KUKA KRL program: f1_Kuka_APT203T03S03.SRC

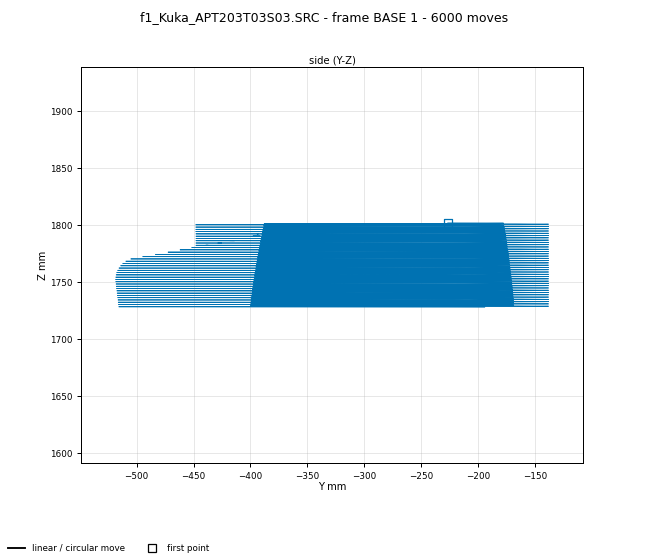
[picture p0: tool path of f1_Kuka_APT203T03S03.SRC in frame BASE 1, 6000 of 6001 moves have a stored position in this frame; points joined in program order, loops and branches not executed]
&ACCESS RVP
&REL 2
&PARAM TEMPLATE = C:\KRC\Roboter\Template\vorgabe
&PARAM EDITMASK = *
DEF f1_Kuka_APT203T03S03()


;FOLD INI;%{PE}%V3.2.0,%MKUKATPBASIS,%CINIT,%VCOMMON,%P
  ;FOLD BAS INI;%{E}%V3.2.0,%MKUKATPBASIS,%CINIT,%VINIT,%P
    GLOBAL INTERRUPT DECL 3 WHEN $STOPMESS==TRUE DO IR_STOPM ( )
    INTERRUPT ON 3
    BAS (#INITMOV,0 )
  ;ENDFOLD (BAS INI)
  ;FOLD USER INI;%{E}%V3.2.0,%MKUKATPUSER,%CINIT,%VINIT,%P
    ;Make your modifications here
  ;ENDFOLD (USER INI)
;ENDFOLD (INI)


;*** Make Null PTP Move
  PTP $pos_act

;*** Auto Load The Correct TOOL Data
  $tool=tool_data[3]

;*** Auto Load The Correct BASE Data
  $base=base_data[1]

  $ADVANCE = 5

;*** Restate Last Velocity
MMPM(30000.0)
SetRPM(6000)
LIN {X 0.049,Y -226.868,Z 1802.195,A 0.000,B 0.000,C 90.000,E1 35.105} C_DIS
LIN {X -0.089,Y -218.794,Z 1802.178,A 0.000,B 0.000,C 90.000,E1 32.084} C_DIS
LIN {X 0.015,Y -211.271,Z 1802.161,A 0.000,B 0.000,C 90.000,E1 28.949} C_DIS
LIN {X -0.003,Y -204.423,Z 1802.143,A 0.000,B 0.000,C 90.000,E1 25.796} C_DIS
LIN {X 0.008,Y -198.407,Z 1802.125,A 0.000,B 0.000,C 90.000,E1 22.589} C_DIS
LIN {X 0.076,Y -193.126,Z 1802.107,A 0.000,B 0.000,C 90.000,E1 19.322} C_DIS
LIN {X -0.059,Y -188.899,Z 1802.089,A 0.000,B 0.000,C 90.000,E1 16.079} C_DIS
LIN {X 0.063,Y -184.696,Z 1802.066,A 0.000,B 0.000,C 90.000,E1 11.895} C_DIS
LIN {X 0.091,Y -181.548,Z 1802.043,A 0.000,B 0.000,C 90.000,E1 7.701} C_DIS
LIN {X -0.028,Y -178.910,Z 1802.010,A 0.000,B 0.000,C 90.000,E1 1.835} C_DIS
LIN {X 0.066,Y -177.903,Z 1801.964,A 0.000,B 0.000,C 90.000,E1 353.571} C_DIS
LIN {X 0.025,Y -178.856,Z 1801.931,A 0.000,B 0.000,C 90.000,E1 347.645} C_DIS
LIN {X -0.075,Y -181.512,Z 1801.894,A 0.000,B 0.000,C 90.000,E1 340.913} C_DIS
LIN {X 0.004,Y -184.682,Z 1801.866,A 0.000,B 0.000,C 90.000,E1 335.845} C_DIS
LIN {X -0.006,Y -188.687,Z 1801.838,A 0.000,B 0.000,C 90.000,E1 330.845} C_DIS
LIN {X 0.009,Y -192.663,Z 1801.815,A 0.000,B 0.000,C 90.000,E1 326.707} C_DIS
LIN {X -0.078,Y -197.668,Z 1801.792,A 0.000,B 0.000,C 90.000,E1 322.637} C_DIS
LIN {X -0.028,Y -202.764,Z 1801.774,A 0.000,B 0.000,C 90.000,E1 319.380} C_DIS
LIN {X -0.078,Y -207.391,Z 1801.761,A 0.000,B 0.000,C 90.000,E1 316.986} C_DIS
LIN {X -0.051,Y -212.928,Z 1801.748,A 0.000,B 0.000,C 90.000,E1 314.595} C_DIS
LIN {X -0.018,Y -217.212,Z 1801.739,A 0.000,B 0.000,C 90.000,E1 313.014} C_DIS
LIN {X -0.070,Y -222.200,Z 1801.730,A 0.000,B 0.000,C 90.000,E1 311.472} C_DIS
LIN {X -0.065,Y -227.868,Z 1801.722,A 0.000,B 0.000,C 90.000,E1 309.930} C_DIS
LIN {X 0.041,Y -234.269,Z 1801.713,A 0.000,B 0.000,C 90.000,E1 308.382} C_DIS
LIN {X 0.068,Y -243.180,Z 1801.703,A 0.000,B 0.000,C 90.000,E1 306.503} C_DIS
LIN {X -0.042,Y -255.247,Z 1801.691,A 0.000,B 0.000,C 90.000,E1 304.326} C_DIS
LIN {X 0.152,Y -268.384,Z 1801.679,A 0.000,B 0.000,C 90.000,E1 302.133} C_DIS
LIN {X -0.140,Y -287.357,Z 1801.663,A 0.000,B 0.000,C 90.000,E1 299.411} C_DIS
LIN {X 0.029,Y -307.519,Z 1801.648,A 0.000,B 0.000,C 90.000,E1 296.693} C_DIS
LIN {X -0.125,Y -323.073,Z 1801.637,A 0.000,B 0.000,C 90.000,E1 294.771} C_DIS
LIN {X 0.059,Y -335.908,Z 1801.629,A 0.000,B 0.000,C 90.000,E1 293.153} C_DIS
LIN {X 0.152,Y -348.343,Z 1801.620,A 0.000,B 0.000,C 90.000,E1 291.589} C_DIS
LIN {X 0.091,Y -355.528,Z 1801.615,A 0.000,B 0.000,C 90.000,E1 290.684} C_DIS
LIN {X -0.107,Y -362.258,Z 1801.610,A 0.000,B 0.000,C 90.000,E1 289.812} C_DIS
LIN {X -0.036,Y -368.425,Z 1801.605,A 0.000,B 0.000,C 90.000,E1 288.906} C_DIS
LIN {X 0.103,Y -373.893,Z 1801.600,A 0.000,B 0.000,C 90.000,E1 288.000} C_DIS
LIN {X -0.069,Y -378.389,Z 1801.595,A 0.000,B 0.000,C 90.000,E1 287.149} C_DIS
LIN {X 0.054,Y -381.951,Z 1801.590,A 0.000,B 0.000,C 90.000,E1 286.260} C_DIS
LIN {X -0.158,Y -384.694,Z 1801.586,A 0.000,B 0.000,C 90.000,E1 285.426} C_DIS
LIN {X -0.008,Y -386.071,Z 1801.582,A 0.000,B 0.000,C 90.000,E1 284.828} C_DIS
LIN {X 0.056,Y -387.102,Z 1801.579,A 0.000,B 0.000,C 90.000,E1 284.245} C_DIS
LIN {X -0.153,Y -387.749,Z 1801.576,A 0.000,B 0.000,C 90.000,E1 283.703} C_DIS
LIN {X -0.072,Y -388.016,Z 1801.573,A 0.000,B 0.000,C 90.000,E1 283.119} C_DIS
LIN {X 0.015,Y -387.896,Z 1801.570,A 0.000,B 0.000,C 90.000,E1 282.535} C_DIS
LIN {X 0.105,Y -387.385,Z 1801.567,A 0.000,B 0.000,C 90.000,E1 281.951} C_DIS
LIN {X -0.184,Y -386.489,Z 1801.563,A 0.000,B 0.000,C 90.000,E1 281.422} C_DIS
LIN {X -0.097,Y -385.220,Z 1801.560,A 0.000,B 0.000,C 90.000,E1 280.838} C_DIS
LIN {X -0.016,Y -383.567,Z 1801.557,A 0.000,B 0.000,C 90.000,E1 280.254} C_DIS
LIN {X 0.084,Y -380.530,Z 1801.552,A 0.000,B 0.000,C 90.000,E1 279.378} C_DIS
LIN {X 0.091,Y -376.860,Z 1801.547,A 0.000,B 0.000,C 90.000,E1 278.511} C_DIS
LIN {X 0.061,Y -374.045,Z 1801.544,A 0.000,B 0.000,C 90.000,E1 277.936} C_DIS
LIN {X 0.013,Y -369.161,Z 1801.539,A 0.000,B 0.000,C 90.000,E1 277.068} C_DIS
LIN {X -0.074,Y -363.286,Z 1801.534,A 0.000,B 0.000,C 90.000,E1 276.201} C_DIS
LIN {X -0.174,Y -358.718,Z 1801.531,A 0.000,B 0.000,C 90.000,E1 275.625} C_DIS
LIN {X 0.056,Y -353.637,Z 1801.528,A 0.000,B 0.000,C 90.000,E1 274.992} C_DIS
LIN {X -0.079,Y -347.942,Z 1801.524,A 0.000,B 0.000,C 90.000,E1 274.416} C_DIS
LIN {X 0.034,Y -342.104,Z 1801.521,A 0.000,B 0.000,C 90.000,E1 273.841} C_DIS
LIN {X 0.014,Y -336.087,Z 1801.518,A 0.000,B 0.000,C 90.000,E1 273.326} C_DIS
LIN {X -0.054,Y -330.045,Z 1801.516,A 0.000,B 0.000,C 90.000,E1 272.865} C_DIS
LIN {X 0.000,Y -323.550,Z 1801.513,A 0.000,B 0.000,C 90.000,E1 272.407} C_DIS
LIN {X -0.005,Y -316.745,Z 1801.511,A 0.000,B 0.000,C 90.000,E1 272.007} C_DIS
LIN {X -0.014,Y -309.834,Z 1801.509,A 0.000,B 0.000,C 90.000,E1 271.661} C_DIS
LIN {X -0.059,Y -302.584,Z 1801.508,A 0.000,B 0.000,C 90.000,E1 271.375} C_DIS
LIN {X -0.122,Y -294.791,Z 1801.506,A 0.000,B 0.000,C 90.000,E1 271.146} C_DIS
LIN {X -0.005,Y -284.000,Z 1801.505,A 0.000,B 0.000,C 90.000,E1 270.859} C_DIS
LIN {X 0.024,Y -272.702,Z 1801.504,A 0.000,B 0.000,C 90.000,E1 270.630} C_DIS
LIN {X -0.103,Y -257.783,Z 1801.502,A 0.000,B 0.000,C 90.000,E1 270.401} C_DIS
LIN {X 0.105,Y -246.724,Z 1801.501,A 0.000,B 0.000,C 90.000,E1 270.229} C_DIS
LIN {X 0.009,Y -235.036,Z 1801.501,A 0.000,B 0.000,C 90.000,E1 270.172} C_DIS
LIN {X -0.015,Y -181.579,Z 1801.501,A 0.000,B 0.000,C 90.000,E1 270.172} C_DIS
LIN {X -0.048,Y -180.792,Z 1801.471,A 0.000,B 0.000,C 90.000,E1 264.780} C_DIS
LIN {X 0.026,Y -178.891,Z 1801.443,A 0.000,B 0.000,C 90.000,E1 259.690} C_DIS
LIN {X -0.068,Y -175.934,Z 1801.414,A 0.000,B 0.000,C 90.000,E1 254.629} C_DIS
LIN {X 0.048,Y -175.381,Z 1801.410,A 0.000,B 0.000,C 90.000,E1 253.740} C_DIS
LIN {X 0.045,Y -172.154,Z 1801.386,A 0.000,B 0.000,C 90.000,E1 249.464} C_DIS
LIN {X 0.082,Y -171.621,Z 1801.381,A 0.000,B 0.000,C 90.000,E1 248.592} C_DIS
LIN {X 0.069,Y -167.843,Z 1801.357,A 0.000,B 0.000,C 90.000,E1 244.280} C_DIS
LIN {X 0.010,Y -166.572,Z 1801.348,A 0.000,B 0.000,C 90.000,E1 242.564} C_DIS
LIN {X -0.004,Y -162.565,Z 1801.323,A 0.000,B 0.000,C 90.000,E1 238.201} C_DIS
LIN {X 0.056,Y -161.246,Z 1801.314,A 0.000,B 0.000,C 90.000,E1 236.421} C_DIS
LIN {X -0.034,Y -157.249,Z 1801.289,A 0.000,B 0.000,C 90.000,E1 232.029} C_DIS
LIN {X 0.013,Y -155.972,Z 1801.279,A 0.000,B 0.000,C 90.000,E1 230.231} C_DIS
LIN {X 0.071,Y -152.226,Z 1801.254,A 0.000,B 0.000,C 90.000,E1 225.729} C_DIS
LIN {X -0.019,Y -150.469,Z 1801.239,A 0.000,B 0.000,C 90.000,E1 223.056} C_DIS
LIN {X 0.001,Y -147.194,Z 1801.214,A 0.000,B 0.000,C 90.000,E1 218.508} C_DIS
LIN {X 0.082,Y -145.213,Z 1801.194,A 0.000,B 0.000,C 90.000,E1 214.818} C_DIS
LIN {X -0.008,Y -142.345,Z 1801.163,A 0.000,B 0.000,C 90.000,E1 209.333} C_DIS
LIN {X 0.045,Y -141.733,Z 1801.153,A 0.000,B 0.000,C 90.000,E1 207.462} C_DIS
LIN {X 0.027,Y -139.483,Z 1801.117,A 0.000,B 0.000,C 90.000,E1 200.972} C_DIS
LIN {X 0.015,Y -138.984,Z 1801.101,A 0.000,B 0.000,C 90.000,E1 198.181} C_DIS
LIN {X -0.023,Y -138.333,Z 1801.054,A 0.000,B 0.000,C 90.000,E1 189.792} C_DIS
LIN {X 0.001,Y -139.425,Z 1801.008,A 0.000,B 0.000,C 90.000,E1 181.375} C_DIS
LIN {X 0.055,Y -141.349,Z 1800.971,A 0.000,B 0.000,C 90.000,E1 174.837} C_DIS
LIN {X 0.032,Y -142.703,Z 1800.956,A 0.000,B 0.000,C 90.000,E1 172.064} C_DIS
LIN {X -0.009,Y -145.073,Z 1800.930,A 0.000,B 0.000,C 90.000,E1 167.465} C_DIS
LIN {X -0.013,Y -147.698,Z 1800.910,A 0.000,B 0.000,C 90.000,E1 163.795} C_DIS
LIN {X 0.019,Y -150.349,Z 1800.890,A 0.000,B 0.000,C 90.000,E1 160.134} C_DIS
LIN {X 0.013,Y -154.604,Z 1800.865,A 0.000,B 0.000,C 90.000,E1 155.613} C_DIS
LIN {X 0.019,Y -158.145,Z 1800.845,A 0.000,B 0.000,C 90.000,E1 152.025} C_DIS
LIN {X 0.065,Y -162.432,Z 1800.825,A 0.000,B 0.000,C 90.000,E1 148.456} C_DIS
LIN {X -0.039,Y -166.691,Z 1800.805,A 0.000,B 0.000,C 90.000,E1 144.975} C_DIS
LIN {X 0.074,Y -171.697,Z 1800.786,A 0.000,B 0.000,C 90.000,E1 141.457} C_DIS
LIN {X 0.008,Y -176.669,Z 1800.767,A 0.000,B 0.000,C 90.000,E1 138.038} C_DIS
LIN {X 0.003,Y -180.965,Z 1800.753,A 0.000,B 0.000,C 90.000,E1 135.486} C_DIS
LIN {X -0.010,Y -186.388,Z 1800.734,A 0.000,B 0.000,C 90.000,E1 132.123} C_DIS
LIN {X -0.070,Y -191.018,Z 1800.720,A 0.000,B 0.000,C 90.000,E1 129.644} C_DIS
LIN {X 0.123,Y -196.798,Z 1800.702,A 0.000,B 0.000,C 90.000,E1 126.297} C_DIS
LIN {X 0.042,Y -200.050,Z 1800.693,A 0.000,B 0.000,C 90.000,E1 124.692} C_DIS
LIN {X 0.036,Y -207.551,Z 1800.670,A 0.000,B 0.000,C 90.000,E1 120.669} C_DIS
LIN {X 0.040,Y -210.761,Z 1800.662,A 0.000,B 0.000,C 90.000,E1 119.077} C_DIS
LIN {X 0.079,Y -213.754,Z 1800.652,A 0.000,B 0.000,C 90.000,E1 117.385} C_DIS
LIN {X 0.074,Y -337.789,Z 1800.652,A 0.000,B 0.000,C 90.000,E1 117.385} C_DIS
LIN {X 0.022,Y -338.618,Z 1800.652,A 0.000,B 0.000,C 90.000,E1 117.385} C_DIS
LIN {X 0.019,Y -343.715,Z 1800.650,A 0.000,B 0.000,C 90.000,E1 117.052} C_DIS
LIN {X -0.141,Y -345.694,Z 1800.648,A 0.000,B 0.000,C 90.000,E1 116.744} C_DIS
LIN {X 0.023,Y -347.535,Z 1800.645,A 0.000,B 0.000,C 90.000,E1 116.104} C_DIS
LIN {X 0.201,Y -349.007,Z 1800.642,A 0.000,B 0.000,C 90.000,E1 115.463} C_DIS
LIN {X -0.076,Y -350.263,Z 1800.638,A 0.000,B 0.000,C 90.000,E1 114.899} C_DIS
LIN {X 0.121,Y -351.140,Z 1800.635,A 0.000,B 0.000,C 90.000,E1 114.259} C_DIS
LIN {X -0.140,Y -351.151,Z 1800.631,A 0.000,B 0.000,C 90.000,E1 113.695} C_DIS
LIN {X 0.111,Y -343.512,Z 1800.608,A 0.000,B 0.000,C 90.000,E1 109.396} C_DIS
LIN {X -0.001,Y -337.369,Z 1800.580,A 0.000,B 0.000,C 90.000,E1 104.411} C_DIS
LIN {X -0.058,Y -337.416,Z 1800.580,A 0.000,B 0.000,C 90.000,E1 104.411} C_DIS
LIN {X -0.125,Y -354.092,Z 1800.568,A 0.000,B 0.000,C 90.000,E1 102.355} C_DIS
LIN {X -0.015,Y -372.554,Z 1800.557,A 0.000,B 0.000,C 90.000,E1 100.310} C_DIS
LIN {X 0.103,Y -391.414,Z 1800.547,A 0.000,B 0.000,C 90.000,E1 98.454} C_DIS
LIN {X 0.110,Y -410.686,Z 1800.538,A 0.000,B 0.000,C 90.000,E1 96.777} C_DIS
LIN {X 0.041,Y -433.088,Z 1800.528,A 0.000,B 0.000,C 90.000,E1 95.049} C_DIS
LIN {X 0.018,Y -438.722,Z 1800.526,A 0.000,B 0.000,C 90.000,E1 94.645} C_DIS
LIN {X -0.017,Y -442.704,Z 1800.524,A 0.000,B 0.000,C 90.000,E1 94.245} C_DIS
LIN {X -0.198,Y -444.401,Z 1800.522,A 0.000,B 0.000,C 90.000,E1 94.012} C_DIS
LIN {X 0.033,Y -445.693,Z 1800.521,A 0.000,B 0.000,C 90.000,E1 93.726} C_DIS
LIN {X -0.045,Y -447.394,Z 1800.518,A 0.000,B 0.000,C 90.000,E1 93.212} C_DIS
LIN {X -0.092,Y -448.057,Z 1800.515,A 0.000,B 0.000,C 90.000,E1 92.694} C_DIS
LIN {X -0.150,Y -447.790,Z 1800.512,A 0.000,B 0.000,C 90.000,E1 92.178} C_DIS
LIN {X -0.188,Y -446.557,Z 1800.509,A 0.000,B 0.000,C 90.000,E1 91.661} C_DIS
LIN {X 0.009,Y -445.523,Z 1800.508,A 0.000,B 0.000,C 90.000,E1 91.375} C_DIS
LIN {X 0.203,Y -444.146,Z 1800.506,A 0.000,B 0.000,C 90.000,E1 91.088} C_DIS
LIN {X -0.166,Y -430.943,Z 1800.495,A 0.000,B 0.000,C 90.000,E1 89.026} C_DIS
LIN {X -0.194,Y -420.924,Z 1800.485,A 0.000,B 0.000,C 90.000,E1 87.421} C_DIS
LIN {X 0.117,Y -409.108,Z 1800.475,A 0.000,B 0.000,C 90.000,E1 85.469} C_DIS
LIN {X -0.190,Y -397.220,Z 1800.464,A 0.000,B 0.000,C 90.000,E1 83.571} C_DIS
LIN {X 0.131,Y -385.260,Z 1800.453,A 0.000,B 0.000,C 90.000,E1 81.546} C_DIS
LIN {X -0.109,Y -373.304,Z 1800.442,A 0.000,B 0.000,C 90.000,E1 79.567} C_DIS
LIN {X 0.097,Y -356.843,Z 1800.426,A 0.000,B 0.000,C 90.000,E1 76.589} C_DIS
LIN {X -0.096,Y -355.062,Z 1800.424,A 0.000,B 0.000,C 90.000,E1 76.284} C_DIS
LIN {X 0.190,Y -355.058,Z 1800.424,A 0.000,B 0.000,C 90.000,E1 76.228} C_DIS
LIN {X -0.055,Y -360.061,Z 1800.412,A 0.000,B 0.000,C 90.000,E1 74.212} C_DIS
LIN {X -0.056,Y -360.127,Z 1800.409,A 0.000,B 0.000,C 90.000,E1 73.614} C_DIS
LIN {X -0.047,Y -359.374,Z 1800.406,A 0.000,B 0.000,C 90.000,E1 73.015} C_DIS
LIN {X -0.038,Y -358.243,Z 1800.402,A 0.000,B 0.000,C 90.000,E1 72.417} C_DIS
LIN {X -0.041,Y -355.353,Z 1800.396,A 0.000,B 0.000,C 90.000,E1 71.221} C_DIS
LIN {X 0.033,Y -351.986,Z 1800.389,A 0.000,B 0.000,C 90.000,E1 70.007} C_DIS
LIN {X -0.070,Y -346.491,Z 1800.379,A 0.000,B 0.000,C 90.000,E1 68.209} C_DIS
LIN {X 0.051,Y -340.599,Z 1800.369,A 0.000,B 0.000,C 90.000,E1 66.357} C_DIS
LIN {X -0.119,Y -334.493,Z 1800.358,A 0.000,B 0.000,C 90.000,E1 64.537} C_DIS
LIN {X -0.105,Y -328.066,Z 1800.348,A 0.000,B 0.000,C 90.000,E1 62.666} C_DIS
LIN {X 0.119,Y -322.241,Z 1800.339,A 0.000,B 0.000,C 90.000,E1 61.051} C_DIS
LIN {X 0.118,Y -315.910,Z 1800.330,A 0.000,B 0.000,C 90.000,E1 59.459} C_DIS
LIN {X 0.068,Y -307.744,Z 1800.320,A 0.000,B 0.000,C 90.000,E1 57.533} C_DIS
LIN {X -0.060,Y -299.204,Z 1800.309,A 0.000,B 0.000,C 90.000,E1 55.595} C_DIS
LIN {X 0.066,Y -290.532,Z 1800.298,A 0.000,B 0.000,C 90.000,E1 53.577} C_DIS
LIN {X -0.007,Y -279.032,Z 1800.283,A 0.000,B 0.000,C 90.000,E1 50.884} C_DIS
LIN {X 0.046,Y -266.931,Z 1800.265,A 0.000,B 0.000,C 90.000,E1 47.757} C_DIS
LIN {X -0.061,Y -255.644,Z 1800.248,A 0.000,B 0.000,C 90.000,E1 44.595} C_DIS
LIN {X 0.060,Y -246.134,Z 1800.232,A 0.000,B 0.000,C 90.000,E1 41.676} C_DIS
LIN {X -0.019,Y -236.966,Z 1800.215,A 0.000,B 0.000,C 90.000,E1 38.749} C_DIS
LIN {X 0.044,Y -226.156,Z 1800.194,A 0.000,B 0.000,C 90.000,E1 34.978} C_DIS
LIN {X 0.009,Y -218.086,Z 1800.177,A 0.000,B 0.000,C 90.000,E1 31.926} C_DIS
LIN {X -0.017,Y -210.578,Z 1800.160,A 0.000,B 0.000,C 90.000,E1 28.821} C_DIS
LIN {X -0.051,Y -203.742,Z 1800.143,A 0.000,B 0.000,C 90.000,E1 25.668} C_DIS
LIN {X -0.056,Y -197.761,Z 1800.125,A 0.000,B 0.000,C 90.000,E1 22.461} C_DIS
LIN {X -0.069,Y -192.520,Z 1800.107,A 0.000,B 0.000,C 90.000,E1 19.214} C_DIS
LIN {X 0.025,Y -188.325,Z 1800.088,A 0.000,B 0.000,C 90.000,E1 15.898} C_DIS
LIN {X -0.055,Y -184.173,Z 1800.065,A 0.000,B 0.000,C 90.000,E1 11.771} C_DIS
LIN {X -0.074,Y -181.053,Z 1800.042,A 0.000,B 0.000,C 90.000,E1 7.587} C_DIS
LIN {X 0.014,Y -178.233,Z 1800.005,A 0.000,B 0.000,C 90.000,E1 0.802} C_DIS
LIN {X 0.050,Y -177.541,Z 1799.964,A 0.000,B 0.000,C 90.000,E1 353.571} C_DIS
LIN {X -0.093,Y -178.758,Z 1799.927,A 0.000,B 0.000,C 90.000,E1 346.825} C_DIS
LIN {X 0.047,Y -181.197,Z 1799.894,A 0.000,B 0.000,C 90.000,E1 340.859} C_DIS
LIN {X -0.056,Y -184.377,Z 1799.866,A 0.000,B 0.000,C 90.000,E1 335.845} C_DIS
LIN {X 0.086,Y -188.424,Z 1799.838,A 0.000,B 0.000,C 90.000,E1 330.795} C_DIS
LIN {X -0.073,Y -192.446,Z 1799.815,A 0.000,B 0.000,C 90.000,E1 326.707} C_DIS
LIN {X 0.108,Y -197.548,Z 1799.792,A 0.000,B 0.000,C 90.000,E1 322.557} C_DIS
LIN {X 0.009,Y -201.339,Z 1799.779,A 0.000,B 0.000,C 90.000,E1 320.150} C_DIS
LIN {X 0.082,Y -205.789,Z 1799.765,A 0.000,B 0.000,C 90.000,E1 317.715} C_DIS
LIN {X 0.079,Y -211.070,Z 1799.752,A 0.000,B 0.000,C 90.000,E1 315.324} C_DIS
LIN {X -0.019,Y -216.221,Z 1799.741,A 0.000,B 0.000,C 90.000,E1 313.380} C_DIS
LIN {X -0.089,Y -221.080,Z 1799.732,A 0.000,B 0.000,C 90.000,E1 311.838} C_DIS
LIN {X 0.075,Y -226.607,Z 1799.724,A 0.000,B 0.000,C 90.000,E1 310.253} C_DIS
LIN {X -0.010,Y -232.839,Z 1799.715,A 0.000,B 0.000,C 90.000,E1 308.749} C_DIS
LIN {X -0.013,Y -241.593,Z 1799.705,A 0.000,B 0.000,C 90.000,E1 306.870} C_DIS
LIN {X -0.012,Y -253.471,Z 1799.693,A 0.000,B 0.000,C 90.000,E1 304.659} C_DIS
LIN {X 0.053,Y -268.761,Z 1799.679,A 0.000,B 0.000,C 90.000,E1 302.133} C_DIS
LIN {X 0.156,Y -287.772,Z 1799.663,A 0.000,B 0.000,C 90.000,E1 299.333} C_DIS
LIN {X -0.030,Y -307.933,Z 1799.648,A 0.000,B 0.000,C 90.000,E1 296.693} C_DIS
LIN {X -0.145,Y -323.490,Z 1799.637,A 0.000,B 0.000,C 90.000,E1 294.771} C_DIS
LIN {X 0.061,Y -336.326,Z 1799.629,A 0.000,B 0.000,C 90.000,E1 293.153} C_DIS
LIN {X 0.162,Y -348.781,Z 1799.620,A 0.000,B 0.000,C 90.000,E1 291.589} C_DIS
LIN {X -0.186,Y -358.269,Z 1799.613,A 0.000,B 0.000,C 90.000,E1 290.429} C_DIS
LIN {X -0.033,Y -364.845,Z 1799.608,A 0.000,B 0.000,C 90.000,E1 289.504} C_DIS
LIN {X 0.070,Y -370.827,Z 1799.603,A 0.000,B 0.000,C 90.000,E1 288.598} C_DIS
LIN {X 0.131,Y -374.380,Z 1799.600,A 0.000,B 0.000,C 90.000,E1 288.000} C_DIS
LIN {X -0.141,Y -377.473,Z 1799.597,A 0.000,B 0.000,C 90.000,E1 287.457} C_DIS
LIN {X 0.078,Y -381.323,Z 1799.592,A 0.000,B 0.000,C 90.000,E1 286.551} C_DIS
LIN {X 0.106,Y -383.392,Z 1799.589,A 0.000,B 0.000,C 90.000,E1 285.969} C_DIS
LIN {X -0.116,Y -385.134,Z 1799.586,A 0.000,B 0.000,C 90.000,E1 285.426} C_DIS
LIN {X 0.038,Y -386.506,Z 1799.582,A 0.000,B 0.000,C 90.000,E1 284.828} C_DIS
LIN {X 0.104,Y -387.522,Z 1799.579,A 0.000,B 0.000,C 90.000,E1 284.245} C_DIS
LIN {X -0.103,Y -388.189,Z 1799.576,A 0.000,B 0.000,C 90.000,E1 283.703} C_DIS
LIN {X -0.020,Y -388.450,Z 1799.573,A 0.000,B 0.000,C 90.000,E1 283.119} C_DIS
LIN {X 0.070,Y -388.333,Z 1799.570,A 0.000,B 0.000,C 90.000,E1 282.535} C_DIS
LIN {X 0.163,Y -387.840,Z 1799.567,A 0.000,B 0.000,C 90.000,E1 281.951} C_DIS
LIN {X -0.124,Y -386.939,Z 1799.563,A 0.000,B 0.000,C 90.000,E1 281.422} C_DIS
LIN {X -0.035,Y -385.696,Z 1799.560,A 0.000,B 0.000,C 90.000,E1 280.838} C_DIS
LIN {X 0.049,Y -384.051,Z 1799.557,A 0.000,B 0.000,C 90.000,E1 280.254} C_DIS
LIN {X 0.153,Y -381.043,Z 1799.552,A 0.000,B 0.000,C 90.000,E1 279.378} C_DIS
LIN {X 0.165,Y -377.390,Z 1799.547,A 0.000,B 0.000,C 90.000,E1 278.511} C_DIS
LIN {X 0.137,Y -374.564,Z 1799.544,A 0.000,B 0.000,C 90.000,E1 277.936} C_DIS
LIN {X 0.092,Y -369.645,Z 1799.539,A 0.000,B 0.000,C 90.000,E1 277.068} C_DIS
LIN {X 0.008,Y -363.751,Z 1799.534,A 0.000,B 0.000,C 90.000,E1 276.201} C_DIS
LIN {X -0.134,Y -356.711,Z 1799.530,A 0.000,B 0.000,C 90.000,E1 275.334} C_DIS
LIN {X 0.110,Y -351.326,Z 1799.526,A 0.000,B 0.000,C 90.000,E1 274.702} C_DIS
LIN {X 0.100,Y -345.622,Z 1799.523,A 0.000,B 0.000,C 90.000,E1 274.131} C_DIS
LIN {X 0.001,Y -339.711,Z 1799.520,A 0.000,B 0.000,C 90.000,E1 273.612} C_DIS
LIN {X 0.107,Y -333.582,Z 1799.517,A 0.000,B 0.000,C 90.000,E1 273.094} C_DIS
LIN {X 0.074,Y -327.302,Z 1799.515,A 0.000,B 0.000,C 90.000,E1 272.636} C_DIS
LIN {X -0.055,Y -320.739,Z 1799.512,A 0.000,B 0.000,C 90.000,E1 272.236} C_DIS
LIN {X 0.073,Y -313.919,Z 1799.510,A 0.000,B 0.000,C 90.000,E1 271.835} C_DIS
LIN {X -0.130,Y -306.791,Z 1799.508,A 0.000,B 0.000,C 90.000,E1 271.547} C_DIS
LIN {X -0.041,Y -299.284,Z 1799.507,A 0.000,B 0.000,C 90.000,E1 271.260} C_DIS
LIN {X -0.136,Y -287.817,Z 1799.505,A 0.000,B 0.000,C 90.000,E1 270.974} C_DIS
LIN {X 0.131,Y -277.007,Z 1799.504,A 0.000,B 0.000,C 90.000,E1 270.688} C_DIS
LIN {X -0.076,Y -257.992,Z 1799.502,A 0.000,B 0.000,C 90.000,E1 270.401} C_DIS
LIN {X 0.118,Y -246.142,Z 1799.501,A 0.000,B 0.000,C 90.000,E1 270.229} C_DIS
LIN {X 0.034,Y -233.356,Z 1799.501,A 0.000,B 0.000,C 90.000,E1 270.172} C_DIS
LIN {X 0.006,Y -181.579,Z 1799.501,A 0.000,B 0.000,C 90.000,E1 270.172} C_DIS
LIN {X -0.023,Y -180.795,Z 1799.471,A 0.000,B 0.000,C 90.000,E1 264.780} C_DIS
LIN {X 0.051,Y -178.894,Z 1799.443,A 0.000,B 0.000,C 90.000,E1 259.690} C_DIS
LIN {X -0.044,Y -175.937,Z 1799.415,A 0.000,B 0.000,C 90.000,E1 254.629} C_DIS
LIN {X 0.070,Y -175.388,Z 1799.410,A 0.000,B 0.000,C 90.000,E1 253.740} C_DIS
LIN {X -0.093,Y -172.159,Z 1799.386,A 0.000,B 0.000,C 90.000,E1 249.518} C_DIS
LIN {X -0.054,Y -171.627,Z 1799.381,A 0.000,B 0.000,C 90.000,E1 248.646} C_DIS
LIN {X -0.058,Y -167.850,Z 1799.357,A 0.000,B 0.000,C 90.000,E1 244.332} C_DIS
LIN {X 0.033,Y -166.579,Z 1799.348,A 0.000,B 0.000,C 90.000,E1 242.564} C_DIS
LIN {X 0.019,Y -162.571,Z 1799.323,A 0.000,B 0.000,C 90.000,E1 238.201} C_DIS
LIN {X 0.078,Y -161.253,Z 1799.314,A 0.000,B 0.000,C 90.000,E1 236.421} C_DIS
LIN {X -0.012,Y -157.255,Z 1799.289,A 0.000,B 0.000,C 90.000,E1 232.029} C_DIS
LIN {X 0.035,Y -155.977,Z 1799.279,A 0.000,B 0.000,C 90.000,E1 230.231} C_DIS
LIN {X 0.092,Y -152.232,Z 1799.254,A 0.000,B 0.000,C 90.000,E1 225.729} C_DIS
LIN {X 0.003,Y -150.474,Z 1799.239,A 0.000,B 0.000,C 90.000,E1 223.056} C_DIS
LIN {X -0.069,Y -147.199,Z 1799.214,A 0.000,B 0.000,C 90.000,E1 218.543} C_DIS
LIN {X -0.015,Y -145.219,Z 1799.194,A 0.000,B 0.000,C 90.000,E1 214.865} C_DIS
LIN {X 0.013,Y -142.348,Z 1799.163,A 0.000,B 0.000,C 90.000,E1 209.333} C_DIS
LIN {X -0.060,Y -141.736,Z 1799.153,A 0.000,B 0.000,C 90.000,E1 207.513} C_DIS
LIN {X 0.048,Y -139.485,Z 1799.117,A 0.000,B 0.000,C 90.000,E1 200.972} C_DIS
LIN {X 0.037,Y -138.986,Z 1799.101,A 0.000,B 0.000,C 90.000,E1 198.181} C_DIS
LIN {X -0.002,Y -138.334,Z 1799.054,A 0.000,B 0.000,C 90.000,E1 189.792} C_DIS
LIN {X 0.022,Y -139.423,Z 1799.008,A 0.000,B 0.000,C 90.000,E1 181.375} C_DIS
LIN {X -0.065,Y -141.345,Z 1798.971,A 0.000,B 0.000,C 90.000,E1 174.894} C_DIS
LIN {X 0.052,Y -142.699,Z 1798.956,A 0.000,B 0.000,C 90.000,E1 172.064} C_DIS
LIN {X 0.012,Y -145.068,Z 1798.930,A 0.000,B 0.000,C 90.000,E1 167.465} C_DIS
LIN {X 0.008,Y -147.693,Z 1798.910,A 0.000,B 0.000,C 90.000,E1 163.795} C_DIS
LIN {X 0.041,Y -150.343,Z 1798.890,A 0.000,B 0.000,C 90.000,E1 160.134} C_DIS
LIN {X 0.035,Y -154.597,Z 1798.865,A 0.000,B 0.000,C 90.000,E1 155.613} C_DIS
LIN {X 0.043,Y -158.136,Z 1798.845,A 0.000,B 0.000,C 90.000,E1 152.025} C_DIS
LIN {X 0.002,Y -162.423,Z 1798.825,A 0.000,B 0.000,C 90.000,E1 148.486} C_DIS
LIN {X -0.016,Y -166.680,Z 1798.805,A 0.000,B 0.000,C 90.000,E1 144.975} C_DIS
LIN {X 0.097,Y -171.686,Z 1798.786,A 0.000,B 0.000,C 90.000,E1 141.457} C_DIS
LIN {X -0.099,Y -176.656,Z 1798.767,A 0.000,B 0.000,C 90.000,E1 138.081} C_DIS
LIN {X 0.028,Y -180.953,Z 1798.753,A 0.000,B 0.000,C 90.000,E1 135.486} C_DIS
LIN {X 0.016,Y -186.375,Z 1798.734,A 0.000,B 0.000,C 90.000,E1 132.123} C_DIS
LIN {X -0.044,Y -191.006,Z 1798.720,A 0.000,B 0.000,C 90.000,E1 129.644} C_DIS
LIN {X -0.009,Y -196.783,Z 1798.702,A 0.000,B 0.000,C 90.000,E1 126.343} C_DIS
LIN {X 0.067,Y -200.035,Z 1798.693,A 0.000,B 0.000,C 90.000,E1 124.692} C_DIS
LIN {X 0.062,Y -207.536,Z 1798.671,A 0.000,B 0.000,C 90.000,E1 120.669} C_DIS
LIN {X 0.066,Y -210.748,Z 1798.662,A 0.000,B 0.000,C 90.000,E1 119.077} C_DIS
LIN {X 0.012,Y -212.937,Z 1798.655,A 0.000,B 0.000,C 90.000,E1 117.847} C_DIS
LIN {X -0.034,Y -337.533,Z 1798.655,A 0.000,B 0.000,C 90.000,E1 117.847} C_DIS
LIN {X 0.219,Y -342.455,Z 1798.654,A 0.000,B 0.000,C 90.000,E1 117.641} C_DIS
LIN {X 0.009,Y -344.383,Z 1798.653,A 0.000,B 0.000,C 90.000,E1 117.513} C_DIS
LIN {X 0.190,Y -347.661,Z 1798.650,A 0.000,B 0.000,C 90.000,E1 117.001} C_DIS
LIN {X -0.115,Y -348.868,Z 1798.648,A 0.000,B 0.000,C 90.000,E1 116.744} C_DIS
LIN {X -0.019,Y -353.641,Z 1798.640,A 0.000,B 0.000,C 90.000,E1 115.207} C_DIS
LIN {X -0.048,Y -357.092,Z 1798.633,A 0.000,B 0.000,C 90.000,E1 114.003} C_DIS
LIN {X 0.046,Y -358.556,Z 1798.630,A 0.000,B 0.000,C 90.000,E1 113.387} C_DIS
LIN {X 0.153,Y -359.679,Z 1798.627,A 0.000,B 0.000,C 90.000,E1 112.770} C_DIS
LIN {X -0.063,Y -360.092,Z 1798.623,A 0.000,B 0.000,C 90.000,E1 112.206} C_DIS
LIN {X 0.185,Y -358.033,Z 1798.617,A 0.000,B 0.000,C 90.000,E1 110.972} C_DIS
LIN {X -0.090,Y -350.927,Z 1798.590,A 0.000,B 0.000,C 90.000,E1 106.205} C_DIS
LIN {X 0.164,Y -347.841,Z 1798.573,A 0.000,B 0.000,C 90.000,E1 103.063} C_DIS
LIN {X 0.107,Y -347.835,Z 1798.573,A 0.000,B 0.000,C 90.000,E1 103.063} C_DIS
LIN {X -0.026,Y -365.342,Z 1798.562,A 0.000,B 0.000,C 90.000,E1 101.074} C_DIS
LIN {X 0.050,Y -384.081,Z 1798.551,A 0.000,B 0.000,C 90.000,E1 99.151} C_DIS
LIN {X 0.101,Y -403.178,Z 1798.541,A 0.000,B 0.000,C 90.000,E1 97.409} C_DIS
LIN {X -0.006,Y -425.444,Z 1798.531,A 0.000,B 0.000,C 90.000,E1 95.625} C_DIS
LIN {X 0.005,Y -439.444,Z 1798.526,A 0.000,B 0.000,C 90.000,E1 94.588} C_DIS
LIN {X -0.110,Y -443.201,Z 1798.523,A 0.000,B 0.000,C 90.000,E1 94.188} C_DIS
LIN {X 0.088,Y -444.820,Z 1798.522,A 0.000,B 0.000,C 90.000,E1 93.898} C_DIS
LIN {X -0.190,Y -446.041,Z 1798.520,A 0.000,B 0.000,C 90.000,E1 93.669} C_DIS
LIN {X 0.205,Y -447.555,Z 1798.517,A 0.000,B 0.000,C 90.000,E1 93.094} C_DIS
LIN {X 0.137,Y -448.062,Z 1798.514,A 0.000,B 0.000,C 90.000,E1 92.579} C_DIS
LIN {X 0.080,Y -447.642,Z 1798.511,A 0.000,B 0.000,C 90.000,E1 92.064} C_DIS
LIN {X 0.041,Y -446.237,Z 1798.509,A 0.000,B 0.000,C 90.000,E1 91.547} C_DIS
LIN {X -0.209,Y -445.097,Z 1798.507,A 0.000,B 0.000,C 90.000,E1 91.318} C_DIS
LIN {X -0.081,Y -440.281,Z 1798.503,A 0.000,B 0.000,C 90.000,E1 90.516} C_DIS
LIN {X 0.186,Y -428.729,Z 1798.493,A 0.000,B 0.000,C 90.000,E1 88.625} C_DIS
LIN {X -0.177,Y -416.978,Z 1798.482,A 0.000,B 0.000,C 90.000,E1 86.788} C_DIS
LIN {X -0.009,Y -406.835,Z 1798.473,A 0.000,B 0.000,C 90.000,E1 85.122} C_DIS
LIN {X 0.034,Y -394.932,Z 1798.462,A 0.000,B 0.000,C 90.000,E1 83.166} C_DIS
LIN {X -0.071,Y -382.980,Z 1798.451,A 0.000,B 0.000,C 90.000,E1 81.197} C_DIS
LIN {X 0.013,Y -369.363,Z 1798.438,A 0.000,B 0.000,C 90.000,E1 78.870} C_DIS
LIN {X -0.124,Y -363.666,Z 1798.433,A 0.000,B 0.000,C 90.000,E1 77.881} C_DIS
LIN {X -0.183,Y -363.619,Z 1798.432,A 0.000,B 0.000,C 90.000,E1 77.881} C_DIS
LIN {X -0.121,Y -368.075,Z 1798.422,A 0.000,B 0.000,C 90.000,E1 75.936} C_DIS
LIN {X -0.076,Y -368.282,Z 1798.418,A 0.000,B 0.000,C 90.000,E1 75.338} C_DIS
LIN {X -0.114,Y -367.539,Z 1798.415,A 0.000,B 0.000,C 90.000,E1 74.755} C_DIS
LIN {X -0.058,Y -366.388,Z 1798.412,A 0.000,B 0.000,C 90.000,E1 74.157} C_DIS
LIN {X 0.043,Y -363.438,Z 1798.405,A 0.000,B 0.000,C 90.000,E1 72.960} C_DIS
LIN {X 0.106,Y -360.002,Z 1798.399,A 0.000,B 0.000,C 90.000,E1 71.764} C_DIS
LIN {X -0.106,Y -354.287,Z 1798.389,A 0.000,B 0.000,C 90.000,E1 70.007} C_DIS
LIN {X 0.157,Y -348.263,Z 1798.379,A 0.000,B 0.000,C 90.000,E1 68.156} C_DIS
LIN {X -0.011,Y -341.980,Z 1798.369,A 0.000,B 0.000,C 90.000,E1 66.357} C_DIS
LIN {X -0.155,Y -335.553,Z 1798.358,A 0.000,B 0.000,C 90.000,E1 64.537} C_DIS
LIN {X 0.164,Y -328.859,Z 1798.348,A 0.000,B 0.000,C 90.000,E1 62.615} C_DIS
LIN {X 0.102,Y -322.819,Z 1798.339,A 0.000,B 0.000,C 90.000,E1 61.051} C_DIS
LIN {X 0.110,Y -316.286,Z 1798.330,A 0.000,B 0.000,C 90.000,E1 59.459} C_DIS
LIN {X 0.013,Y -309.279,Z 1798.322,A 0.000,B 0.000,C 90.000,E1 57.867} C_DIS
LIN {X 0.137,Y -301.981,Z 1798.313,A 0.000,B 0.000,C 90.000,E1 56.215} C_DIS
LIN {X 0.069,Y -291.650,Z 1798.300,A 0.000,B 0.000,C 90.000,E1 53.909} C_DIS
LIN {X -0.145,Y -280.070,Z 1798.285,A 0.000,B 0.000,C 90.000,E1 51.251} C_DIS
LIN {X 0.148,Y -267.887,Z 1798.267,A 0.000,B 0.000,C 90.000,E1 48.081} C_DIS
LIN {X -0.092,Y -255.287,Z 1798.248,A 0.000,B 0.000,C 90.000,E1 44.595} C_DIS
LIN {X 0.023,Y -244.632,Z 1798.229,A 0.000,B 0.000,C 90.000,E1 41.310} C_DIS
LIN {X -0.089,Y -235.487,Z 1798.213,A 0.000,B 0.000,C 90.000,E1 38.382} C_DIS
LIN {X -0.010,Y -225.770,Z 1798.194,A 0.000,B 0.000,C 90.000,E1 34.978} C_DIS
LIN {X -0.054,Y -217.673,Z 1798.177,A 0.000,B 0.000,C 90.000,E1 31.926} C_DIS
LIN {X -0.088,Y -210.155,Z 1798.160,A 0.000,B 0.000,C 90.000,E1 28.821} C_DIS
LIN {X -0.041,Y -203.314,Z 1798.142,A 0.000,B 0.000,C 90.000,E1 25.643} C_DIS
LIN {X 0.039,Y -197.327,Z 1798.125,A 0.000,B 0.000,C 90.000,E1 22.408} C_DIS
LIN {X 0.081,Y -192.108,Z 1798.106,A 0.000,B 0.000,C 90.000,E1 19.141} C_DIS
LIN {X -0.077,Y -187.894,Z 1798.088,A 0.000,B 0.000,C 90.000,E1 15.898} C_DIS
LIN {X 0.012,Y -183.763,Z 1798.065,A 0.000,B 0.000,C 90.000,E1 11.715} C_DIS
LIN {X -0.018,Y -180.648,Z 1798.042,A 0.000,B 0.000,C 90.000,E1 7.530} C_DIS
LIN {X 0.050,Y -177.848,Z 1798.004,A 0.000,B 0.000,C 90.000,E1 0.745} C_DIS
LIN {X 0.002,Y -177.151,Z 1797.969,A 0.000,B 0.000,C 90.000,E1 354.432} C_DIS
LIN {X 0.054,Y -177.927,Z 1797.936,A 0.000,B 0.000,C 90.000,E1 348.465} C_DIS
LIN {X 0.017,Y -180.038,Z 1797.903,A 0.000,B 0.000,C 90.000,E1 342.543} C_DIS
LIN {X 0.009,Y -182.949,Z 1797.875,A 0.000,B 0.000,C 90.000,E1 337.486} C_DIS
LIN {X -0.073,Y -186.718,Z 1797.847,A 0.000,B 0.000,C 90.000,E1 332.487} C_DIS
LIN {X -0.054,Y -190.505,Z 1797.824,A 0.000,B 0.000,C 90.000,E1 328.329} C_DIS
LIN {X 0.003,Y -195.191,Z 1797.801,A 0.000,B 0.000,C 90.000,E1 324.196} C_DIS
LIN {X 0.028,Y -199.922,Z 1797.783,A 0.000,B 0.000,C 90.000,E1 320.928} C_DIS
LIN {X -0.014,Y -205.815,Z 1797.765,A 0.000,B 0.000,C 90.000,E1 317.715} C_DIS
LIN {X -0.018,Y -211.162,Z 1797.752,A 0.000,B 0.000,C 90.000,E1 315.324} C_DIS
LIN {X 0.045,Y -216.373,Z 1797.741,A 0.000,B 0.000,C 90.000,E1 313.338} C_DIS
LIN {X 0.132,Y -221.231,Z 1797.732,A 0.000,B 0.000,C 90.000,E1 311.757} C_DIS
LIN {X -0.017,Y -226.818,Z 1797.724,A 0.000,B 0.000,C 90.000,E1 310.253} C_DIS
LIN {X -0.103,Y -233.069,Z 1797.715,A 0.000,B 0.000,C 90.000,E1 308.749} C_DIS
LIN {X -0.105,Y -241.871,Z 1797.705,A 0.000,B 0.000,C 90.000,E1 306.870} C_DIS
LIN {X 0.106,Y -253.777,Z 1797.692,A 0.000,B 0.000,C 90.000,E1 304.612} C_DIS
LIN {X -0.036,Y -269.119,Z 1797.678,A 0.000,B 0.000,C 90.000,E1 302.133} C_DIS
LIN {X 0.070,Y -288.159,Z 1797.663,A 0.000,B 0.000,C 90.000,E1 299.333} C_DIS
LIN {X 0.005,Y -308.193,Z 1797.648,A 0.000,B 0.000,C 90.000,E1 296.693} C_DIS
LIN {X -0.034,Y -323.706,Z 1797.638,A 0.000,B 0.000,C 90.000,E1 294.771} C_DIS
LIN {X -0.145,Y -336.615,Z 1797.629,A 0.000,B 0.000,C 90.000,E1 293.206} C_DIS
LIN {X -0.052,Y -349.071,Z 1797.620,A 0.000,B 0.000,C 90.000,E1 291.642} C_DIS
LIN {X -0.069,Y -358.593,Z 1797.613,A 0.000,B 0.000,C 90.000,E1 290.429} C_DIS
LIN {X 0.090,Y -365.225,Z 1797.608,A 0.000,B 0.000,C 90.000,E1 289.504} C_DIS
LIN {X 0.113,Y -369.304,Z 1797.605,A 0.000,B 0.000,C 90.000,E1 288.906} C_DIS
LIN {X -0.093,Y -374.760,Z 1797.600,A 0.000,B 0.000,C 90.000,E1 288.055} C_DIS
LIN {X -0.006,Y -377.845,Z 1797.597,A 0.000,B 0.000,C 90.000,E1 287.457} C_DIS
LIN {X 0.104,Y -380.521,Z 1797.594,A 0.000,B 0.000,C 90.000,E1 286.858} C_DIS
LIN {X -0.120,Y -383.785,Z 1797.589,A 0.000,B 0.000,C 90.000,E1 286.024} C_DIS
LIN {X 0.031,Y -385.527,Z 1797.586,A 0.000,B 0.000,C 90.000,E1 285.426} C_DIS
LIN {X 0.187,Y -386.916,Z 1797.583,A 0.000,B 0.000,C 90.000,E1 284.828} C_DIS
LIN {X -0.121,Y -387.921,Z 1797.579,A 0.000,B 0.000,C 90.000,E1 284.300} C_DIS
LIN {X 0.051,Y -388.586,Z 1797.576,A 0.000,B 0.000,C 90.000,E1 283.703} C_DIS
LIN {X 0.137,Y -388.875,Z 1797.573,A 0.000,B 0.000,C 90.000,E1 283.119} C_DIS
LIN {X -0.149,Y -388.752,Z 1797.570,A 0.000,B 0.000,C 90.000,E1 282.591} C_DIS
LIN {X -0.055,Y -388.267,Z 1797.567,A 0.000,B 0.000,C 90.000,E1 282.007} C_DIS
LIN {X 0.041,Y -387.404,Z 1797.563,A 0.000,B 0.000,C 90.000,E1 281.422} C_DIS
LIN {X 0.132,Y -386.163,Z 1797.560,A 0.000,B 0.000,C 90.000,E1 280.838} C_DIS
LIN {X -0.161,Y -384.584,Z 1797.557,A 0.000,B 0.000,C 90.000,E1 280.310} C_DIS
LIN {X -0.114,Y -381.605,Z 1797.552,A 0.000,B 0.000,C 90.000,E1 279.443} C_DIS
LIN {X -0.034,Y -378.011,Z 1797.548,A 0.000,B 0.000,C 90.000,E1 278.568} C_DIS
LIN {X -0.051,Y -373.605,Z 1797.543,A 0.000,B 0.000,C 90.000,E1 277.701} C_DIS
LIN {X -0.100,Y -368.347,Z 1797.538,A 0.000,B 0.000,C 90.000,E1 276.834} C_DIS
LIN {X -0.172,Y -364.296,Z 1797.535,A 0.000,B 0.000,C 90.000,E1 276.258} C_DIS
LIN {X 0.094,Y -359.756,Z 1797.531,A 0.000,B 0.000,C 90.000,E1 275.625} C_DIS
LIN {X -0.026,Y -354.649,Z 1797.528,A 0.000,B 0.000,C 90.000,E1 275.049} C_DIS
LIN {X -0.109,Y -349.018,Z 1797.525,A 0.000,B 0.000,C 90.000,E1 274.473} C_DIS
LIN {X -0.017,Y -343.156,Z 1797.522,A 0.000,B 0.000,C 90.000,E1 273.898} C_DIS
LIN {X -0.049,Y -337.134,Z 1797.519,A 0.000,B 0.000,C 90.000,E1 273.383} C_DIS
LIN {X -0.159,Y -330.929,Z 1797.516,A 0.000,B 0.000,C 90.000,E1 272.922} C_DIS
LIN {X -0.077,Y -324.541,Z 1797.514,A 0.000,B 0.000,C 90.000,E1 272.465} C_DIS
LIN {X -0.118,Y -317.728,Z 1797.511,A 0.000,B 0.000,C 90.000,E1 272.064} C_DIS
LIN {X 0.142,Y -310.742,Z 1797.509,A 0.000,B 0.000,C 90.000,E1 271.661} C_DIS
LIN {X 0.060,Y -303.297,Z 1797.508,A 0.000,B 0.000,C 90.000,E1 271.375} C_DIS
LIN {X -0.002,Y -295.630,Z 1797.506,A 0.000,B 0.000,C 90.000,E1 271.146} C_DIS
LIN {X 0.084,Y -284.624,Z 1797.505,A 0.000,B 0.000,C 90.000,E1 270.859} C_DIS
LIN {X 0.084,Y -273.250,Z 1797.504,A 0.000,B 0.000,C 90.000,E1 270.630} C_DIS
LIN {X -0.034,Y -258.206,Z 1797.502,A 0.000,B 0.000,C 90.000,E1 270.401} C_DIS
LIN {X -0.084,Y -246.394,Z 1797.501,A 0.000,B 0.000,C 90.000,E1 270.286} C_DIS
LIN {X 0.078,Y -232.148,Z 1797.501,A 0.000,B 0.000,C 90.000,E1 270.172} C_DIS
LIN {X 0.042,Y -181.579,Z 1797.501,A 0.000,B 0.000,C 90.000,E1 270.172} C_DIS
LIN {X 0.015,Y -180.800,Z 1797.471,A 0.000,B 0.000,C 90.000,E1 264.780} C_DIS
LIN {X -0.087,Y -178.899,Z 1797.443,A 0.000,B 0.000,C 90.000,E1 259.746} C_DIS
LIN {X -0.006,Y -175.942,Z 1797.415,A 0.000,B 0.000,C 90.000,E1 254.629} C_DIS
LIN {X -0.060,Y -175.398,Z 1797.410,A 0.000,B 0.000,C 90.000,E1 253.795} C_DIS
LIN {X -0.056,Y -172.167,Z 1797.386,A 0.000,B 0.000,C 90.000,E1 249.518} C_DIS
LIN {X -0.017,Y -171.635,Z 1797.381,A 0.000,B 0.000,C 90.000,E1 248.646} C_DIS
LIN {X -0.022,Y -167.859,Z 1797.357,A 0.000,B 0.000,C 90.000,E1 244.332} C_DIS
LIN {X -0.078,Y -166.591,Z 1797.348,A 0.000,B 0.000,C 90.000,E1 242.615} C_DIS
LIN {X 0.055,Y -162.581,Z 1797.323,A 0.000,B 0.000,C 90.000,E1 238.201} C_DIS
LIN {X -0.109,Y -161.264,Z 1797.314,A 0.000,B 0.000,C 90.000,E1 236.501} C_DIS
LIN {X 0.024,Y -157.265,Z 1797.289,A 0.000,B 0.000,C 90.000,E1 232.029} C_DIS
LIN {X -0.050,Y -155.985,Z 1797.279,A 0.000,B 0.000,C 90.000,E1 230.275} C_DIS
LIN {X -0.088,Y -152.241,Z 1797.254,A 0.000,B 0.000,C 90.000,E1 225.810} C_DIS
LIN {X 0.037,Y -150.483,Z 1797.239,A 0.000,B 0.000,C 90.000,E1 223.056} C_DIS
LIN {X -0.036,Y -147.207,Z 1797.214,A 0.000,B 0.000,C 90.000,E1 218.543} C_DIS
LIN {X -0.065,Y -145.227,Z 1797.194,A 0.000,B 0.000,C 90.000,E1 214.898} C_DIS
LIN {X 0.046,Y -142.353,Z 1797.163,A 0.000,B 0.000,C 90.000,E1 209.333} C_DIS
LIN {X -0.026,Y -141.741,Z 1797.153,A 0.000,B 0.000,C 90.000,E1 207.513} C_DIS
LIN {X 0.081,Y -139.488,Z 1797.117,A 0.000,B 0.000,C 90.000,E1 200.972} C_DIS
LIN {X 0.069,Y -138.990,Z 1797.101,A 0.000,B 0.000,C 90.000,E1 198.181} C_DIS
LIN {X 0.030,Y -138.336,Z 1797.054,A 0.000,B 0.000,C 90.000,E1 189.792} C_DIS
LIN {X 0.055,Y -139.419,Z 1797.008,A 0.000,B 0.000,C 90.000,E1 181.375} C_DIS
LIN {X -0.032,Y -141.339,Z 1796.972,A 0.000,B 0.000,C 90.000,E1 174.894} C_DIS
LIN {X -0.075,Y -142.695,Z 1796.956,A 0.000,B 0.000,C 90.000,E1 172.129} C_DIS
LIN {X 0.045,Y -145.060,Z 1796.930,A 0.000,B 0.000,C 90.000,E1 167.465} C_DIS
LIN {X 0.042,Y -147.685,Z 1796.910,A 0.000,B 0.000,C 90.000,E1 163.795} C_DIS
LIN {X -0.065,Y -150.332,Z 1796.890,A 0.000,B 0.000,C 90.000,E1 160.188} C_DIS
LIN {X 0.006,Y -153.750,Z 1796.870,A 0.000,B 0.000,C 90.000,E1 156.538} C_DIS
LIN {X -0.003,Y -157.162,Z 1796.850,A 0.000,B 0.000,C 90.000,E1 152.948} C_DIS
LIN {X -0.069,Y -161.316,Z 1796.830,A 0.000,B 0.000,C 90.000,E1 149.410} C_DIS
LIN {X -0.053,Y -164.430,Z 1796.815,A 0.000,B 0.000,C 90.000,E1 146.755} C_DIS
LIN {X 0.079,Y -169.116,Z 1796.796,A 0.000,B 0.000,C 90.000,E1 143.210} C_DIS
LIN {X -0.106,Y -171.670,Z 1796.786,A 0.000,B 0.000,C 90.000,E1 141.537} C_DIS
LIN {X -0.061,Y -176.637,Z 1796.767,A 0.000,B 0.000,C 90.000,E1 138.081} C_DIS
LIN {X 0.066,Y -180.934,Z 1796.753,A 0.000,B 0.000,C 90.000,E1 135.486} C_DIS
LIN {X 0.055,Y -186.354,Z 1796.734,A 0.000,B 0.000,C 90.000,E1 132.123} C_DIS
LIN {X -0.004,Y -190.986,Z 1796.720,A 0.000,B 0.000,C 90.000,E1 129.644} C_DIS
LIN {X -0.086,Y -196.761,Z 1796.702,A 0.000,B 0.000,C 90.000,E1 126.377} C_DIS
LIN {X -0.055,Y -200.010,Z 1796.693,A 0.000,B 0.000,C 90.000,E1 124.739} C_DIS
LIN {X -0.074,Y -207.512,Z 1796.671,A 0.000,B 0.000,C 90.000,E1 120.718} C_DIS
LIN {X 0.109,Y -210.729,Z 1796.662,A 0.000,B 0.000,C 90.000,E1 119.077} C_DIS
LIN {X 0.044,Y -212.368,Z 1796.656,A 0.000,B 0.000,C 90.000,E1 118.153} C_DIS
LIN {X 0.021,Y -338.002,Z 1796.656,A 0.000,B 0.000,C 90.000,E1 118.153} C_DIS
LIN {X -0.078,Y -339.237,Z 1796.656,A 0.000,B 0.000,C 90.000,E1 118.153} C_DIS
LIN {X -0.081,Y -344.876,Z 1796.655,A 0.000,B 0.000,C 90.000,E1 117.847} C_DIS
LIN {X 0.079,Y -347.479,Z 1796.653,A 0.000,B 0.000,C 90.000,E1 117.513} C_DIS
LIN {X 0.086,Y -349.229,Z 1796.651,A 0.000,B 0.000,C 90.000,E1 117.206} C_DIS
LIN {X -0.015,Y -352.631,Z 1796.646,A 0.000,B 0.000,C 90.000,E1 116.309} C_DIS
LIN {X -0.117,Y -359.027,Z 1796.636,A 0.000,B 0.000,C 90.000,E1 114.515} C_DIS
LIN {X -0.213,Y -363.080,Z 1796.629,A 0.000,B 0.000,C 90.000,E1 113.334} C_DIS
LIN {X 0.070,Y -366.687,Z 1796.623,A 0.000,B 0.000,C 90.000,E1 112.099} C_DIS
LIN {X -0.111,Y -368.135,Z 1796.620,A 0.000,B 0.000,C 90.000,E1 111.535} C_DIS
LIN {X 0.059,Y -369.079,Z 1796.616,A 0.000,B 0.000,C 90.000,E1 110.918} C_DIS
LIN {X -0.108,Y -368.782,Z 1796.613,A 0.000,B 0.000,C 90.000,E1 110.355} C_DIS
LIN {X 0.023,Y -361.951,Z 1796.587,A 0.000,B 0.000,C 90.000,E1 105.607} C_DIS
LIN {X 0.071,Y -358.490,Z 1796.566,A 0.000,B 0.000,C 90.000,E1 101.827} C_DIS
LIN {X 0.013,Y -358.487,Z 1796.566,A 0.000,B 0.000,C 90.000,E1 101.827} C_DIS
LIN {X 0.090,Y -375.243,Z 1796.556,A 0.000,B 0.000,C 90.000,E1 100.018} C_DIS
LIN {X -0.028,Y -394.198,Z 1796.546,A 0.000,B 0.000,C 90.000,E1 98.219} C_DIS
LIN {X 0.166,Y -416.287,Z 1796.535,A 0.000,B 0.000,C 90.000,E1 96.315} C_DIS
LIN {X -0.005,Y -438.754,Z 1796.526,A 0.000,B 0.000,C 90.000,E1 94.645} C_DIS
LIN {X -0.043,Y -442.715,Z 1796.524,A 0.000,B 0.000,C 90.000,E1 94.245} C_DIS
LIN {X 0.210,Y -444.409,Z 1796.522,A 0.000,B 0.000,C 90.000,E1 93.955} C_DIS
LIN {X -0.011,Y -445.698,Z 1796.521,A 0.000,B 0.000,C 90.000,E1 93.726} C_DIS
LIN {X -0.089,Y -447.382,Z 1796.518,A 0.000,B 0.000,C 90.000,E1 93.212} C_DIS
LIN {X -0.135,Y -448.031,Z 1796.515,A 0.000,B 0.000,C 90.000,E1 92.694} C_DIS
LIN {X -0.194,Y -447.750,Z 1796.512,A 0.000,B 0.000,C 90.000,E1 92.178} C_DIS
LIN {X 0.214,Y -446.504,Z 1796.509,A 0.000,B 0.000,C 90.000,E1 91.604} C_DIS
LIN {X -0.036,Y -445.461,Z 1796.508,A 0.000,B 0.000,C 90.000,E1 91.375} C_DIS
LIN {X 0.159,Y -444.073,Z 1796.506,A 0.000,B 0.000,C 90.000,E1 91.088} C_DIS
LIN {X -0.210,Y -430.870,Z 1796.494,A 0.000,B 0.000,C 90.000,E1 89.026} C_DIS
LIN {X 0.181,Y -420.852,Z 1796.485,A 0.000,B 0.000,C 90.000,E1 87.364} C_DIS
LIN {X 0.072,Y -409.034,Z 1796.475,A 0.000,B 0.000,C 90.000,E1 85.469} C_DIS
LIN {X 0.159,Y -397.147,Z 1796.464,A 0.000,B 0.000,C 90.000,E1 83.514} C_DIS
LIN {X 0.086,Y -385.185,Z 1796.453,A 0.000,B 0.000,C 90.000,E1 81.546} C_DIS
LIN {X 0.057,Y -372.432,Z 1796.441,A 0.000,B 0.000,C 90.000,E1 79.398} C_DIS
LIN {X -0.003,Y -372.420,Z 1796.441,A 0.000,B 0.000,C 90.000,E1 79.398} C_DIS
LIN {X -0.145,Y -375.837,Z 1796.432,A 0.000,B 0.000,C 90.000,E1 77.813} C_DIS
LIN {X -0.138,Y -376.736,Z 1796.429,A 0.000,B 0.000,C 90.000,E1 77.229} C_DIS
LIN {X -0.124,Y -376.246,Z 1796.426,A 0.000,B 0.000,C 90.000,E1 76.645} C_DIS
LIN {X -0.017,Y -375.175,Z 1796.422,A 0.000,B 0.000,C 90.000,E1 76.047} C_DIS
LIN {X -0.004,Y -373.794,Z 1796.419,A 0.000,B 0.000,C 90.000,E1 75.463} C_DIS
LIN {X 0.087,Y -370.541,Z 1796.413,A 0.000,B 0.000,C 90.000,E1 74.283} C_DIS
LIN {X -0.113,Y -366.879,Z 1796.406,A 0.000,B 0.000,C 90.000,E1 73.142} C_DIS
LIN {X 0.030,Y -360.943,Z 1796.396,A 0.000,B 0.000,C 90.000,E1 71.348} C_DIS
LIN {X -0.046,Y -354.633,Z 1796.386,A 0.000,B 0.000,C 90.000,E1 69.571} C_DIS
LIN {X 0.095,Y -348.180,Z 1796.376,A 0.000,B 0.000,C 90.000,E1 67.741} C_DIS
LIN {X 0.055,Y -340.405,Z 1796.365,A 0.000,B 0.000,C 90.000,E1 65.613} C_DIS
LIN {X 0.002,Y -333.628,Z 1796.354,A 0.000,B 0.000,C 90.000,E1 63.768} C_DIS
LIN {X -0.133,Y -327.711,Z 1796.346,A 0.000,B 0.000,C 90.000,E1 62.231} C_DIS
LIN {X -0.051,Y -321.329,Z 1796.337,A 0.000,B 0.000,C 90.000,E1 60.639} C_DIS
LIN {X 0.211,Y -314.464,Z 1796.328,A 0.000,B 0.000,C 90.000,E1 58.997} C_DIS
LIN {X -0.131,Y -305.625,Z 1796.317,A 0.000,B 0.000,C 90.000,E1 57.120} C_DIS
LIN {X -0.108,Y -293.697,Z 1796.303,A 0.000,B 0.000,C 90.000,E1 54.482} C_DIS
LIN {X -0.139,Y -280.576,Z 1796.286,A 0.000,B 0.000,C 90.000,E1 51.457} C_DIS
LIN {X -0.005,Y -268.348,Z 1796.268,A 0.000,B 0.000,C 90.000,E1 48.324} C_DIS
LIN {X -0.080,Y -256.903,Z 1796.251,A 0.000,B 0.000,C 90.000,E1 45.162} C_DIS
LIN {X -0.107,Y -247.317,Z 1796.235,A 0.000,B 0.000,C 90.000,E1 42.285} C_DIS
LIN {X -0.017,Y -236.919,Z 1796.216,A 0.000,B 0.000,C 90.000,E1 38.955} C_DIS
LIN {X 0.085,Y -228.133,Z 1796.200,A 0.000,B 0.000,C 90.000,E1 35.931} C_DIS
LIN {X 0.092,Y -219.834,Z 1796.183,A 0.000,B 0.000,C 90.000,E1 32.880} C_DIS
LIN {X 0.029,Y -212.144,Z 1796.166,A 0.000,B 0.000,C 90.000,E1 29.795} C_DIS
LIN {X -0.061,Y -205.053,Z 1796.148,A 0.000,B 0.000,C 90.000,E1 26.668} C_DIS
LIN {X -0.040,Y -198.768,Z 1796.130,A 0.000,B 0.000,C 90.000,E1 23.462} C_DIS
LIN {X 0.044,Y -193.302,Z 1796.112,A 0.000,B 0.000,C 90.000,E1 20.194} C_DIS
LIN {X 0.035,Y -188.743,Z 1796.094,A 0.000,B 0.000,C 90.000,E1 16.913} C_DIS
LIN {X 0.012,Y -184.339,Z 1796.071,A 0.000,B 0.000,C 90.000,E1 12.771} C_DIS
LIN {X 0.060,Y -180.946,Z 1796.048,A 0.000,B 0.000,C 90.000,E1 8.568} C_DIS
LIN {X -0.062,Y -178.035,Z 1796.015,A 0.000,B 0.000,C 90.000,E1 2.694} C_DIS
LIN {X -0.089,Y -176.851,Z 1795.979,A 0.000,B 0.000,C 90.000,E1 356.159} C_DIS
LIN {X -0.054,Y -177.417,Z 1795.941,A 0.000,B 0.000,C 90.000,E1 349.342} C_DIS
LIN {X 0.014,Y -179.337,Z 1795.908,A 0.000,B 0.000,C 90.000,E1 343.378} C_DIS
LIN {X 0.094,Y -182.114,Z 1795.880,A 0.000,B 0.000,C 90.000,E1 338.284} C_DIS
LIN {X 0.077,Y -185.736,Z 1795.852,A 0.000,B 0.000,C 90.000,E1 333.256} C_DIS
LIN {X -0.023,Y -189.470,Z 1795.828,A 0.000,B 0.000,C 90.000,E1 329.125} C_DIS
LIN {X 0.058,Y -194.004,Z 1795.806,A 0.000,B 0.000,C 90.000,E1 324.975} C_DIS
LIN {X -0.069,Y -198.559,Z 1795.787,A 0.000,B 0.000,C 90.000,E1 321.743} C_DIS
LIN {X -0.022,Y -202.707,Z 1795.774,A 0.000,B 0.000,C 90.000,E1 319.299} C_DIS
LIN {X -0.073,Y -207.558,Z 1795.760,A 0.000,B 0.000,C 90.000,E1 316.905} C_DIS
LIN {X -0.042,Y -213.278,Z 1795.747,A 0.000,B 0.000,C 90.000,E1 314.514} C_DIS
LIN {X 0.002,Y -217.681,Z 1795.739,A 0.000,B 0.000,C 90.000,E1 312.933} C_DIS
LIN {X -0.046,Y -222.732,Z 1795.730,A 0.000,B 0.000,C 90.000,E1 311.391} C_DIS
LIN {X -0.034,Y -228.542,Z 1795.721,A 0.000,B 0.000,C 90.000,E1 309.850} C_DIS
LIN {X 0.081,Y -234.997,Z 1795.713,A 0.000,B 0.000,C 90.000,E1 308.302} C_DIS
LIN {X -0.024,Y -244.053,Z 1795.703,A 0.000,B 0.000,C 90.000,E1 306.457} C_DIS
LIN {X 0.027,Y -256.191,Z 1795.690,A 0.000,B 0.000,C 90.000,E1 304.246} C_DIS
LIN {X 0.077,Y -274.071,Z 1795.674,A 0.000,B 0.000,C 90.000,E1 301.386} C_DIS
LIN {X -0.056,Y -291.047,Z 1795.661,A 0.000,B 0.000,C 90.000,E1 298.999} C_DIS
LIN {X -0.163,Y -311.392,Z 1795.646,A 0.000,B 0.000,C 90.000,E1 296.360} C_DIS
LIN {X 0.038,Y -327.112,Z 1795.635,A 0.000,B 0.000,C 90.000,E1 294.387} C_DIS
LIN {X 0.007,Y -337.427,Z 1795.629,A 0.000,B 0.000,C 90.000,E1 293.131} C_DIS
LIN {X -0.012,Y -349.883,Z 1795.620,A 0.000,B 0.000,C 90.000,E1 291.589} C_DIS
LIN {X -0.015,Y -359.407,Z 1795.613,A 0.000,B 0.000,C 90.000,E1 290.375} C_DIS
LIN {X 0.154,Y -366.030,Z 1795.608,A 0.000,B 0.000,C 90.000,E1 289.450} C_DIS
LIN {X -0.165,Y -370.096,Z 1795.605,A 0.000,B 0.000,C 90.000,E1 288.906} C_DIS
LIN {X -0.012,Y -375.477,Z 1795.600,A 0.000,B 0.000,C 90.000,E1 288.000} C_DIS
LIN {X 0.082,Y -378.533,Z 1795.597,A 0.000,B 0.000,C 90.000,E1 287.402} C_DIS
LIN {X -0.167,Y -381.173,Z 1795.594,A 0.000,B 0.000,C 90.000,E1 286.858} C_DIS
LIN {X -0.017,Y -384.387,Z 1795.589,A 0.000,B 0.000,C 90.000,E1 285.969} C_DIS
LIN {X 0.139,Y -386.074,Z 1795.585,A 0.000,B 0.000,C 90.000,E1 285.371} C_DIS
LIN {X -0.075,Y -387.430,Z 1795.582,A 0.000,B 0.000,C 90.000,E1 284.828} C_DIS
LIN {X -0.003,Y -388.424,Z 1795.579,A 0.000,B 0.000,C 90.000,E1 284.245} C_DIS
LIN {X 0.173,Y -389.019,Z 1795.576,A 0.000,B 0.000,C 90.000,E1 283.647} C_DIS
LIN {X -0.116,Y -389.269,Z 1795.573,A 0.000,B 0.000,C 90.000,E1 283.119} C_DIS
LIN {X -0.020,Y -389.132,Z 1795.570,A 0.000,B 0.000,C 90.000,E1 282.535} C_DIS
LIN {X 0.077,Y -388.607,Z 1795.566,A 0.000,B 0.000,C 90.000,E1 281.951} C_DIS
LIN {X -0.205,Y -387.739,Z 1795.563,A 0.000,B 0.000,C 90.000,E1 281.422} C_DIS
LIN {X -0.110,Y -386.500,Z 1795.560,A 0.000,B 0.000,C 90.000,E1 280.838} C_DIS
LIN {X -0.022,Y -384.926,Z 1795.557,A 0.000,B 0.000,C 90.000,E1 280.254} C_DIS
LIN {X 0.090,Y -381.921,Z 1795.552,A 0.000,B 0.000,C 90.000,E1 279.378} C_DIS
LIN {X 0.111,Y -378.277,Z 1795.547,A 0.000,B 0.000,C 90.000,E1 278.511} C_DIS
LIN {X 0.095,Y -373.833,Z 1795.543,A 0.000,B 0.000,C 90.000,E1 277.644} C_DIS
LIN {X 0.047,Y -368.514,Z 1795.538,A 0.000,B 0.000,C 90.000,E1 276.777} C_DIS
LIN {X -0.026,Y -364.433,Z 1795.534,A 0.000,B 0.000,C 90.000,E1 276.201} C_DIS
LIN {X -0.161,Y -357.306,Z 1795.530,A 0.000,B 0.000,C 90.000,E1 275.334} C_DIS
LIN {X 0.074,Y -349.009,Z 1795.525,A 0.000,B 0.000,C 90.000,E1 274.416} C_DIS
LIN {X -0.141,Y -343.164,Z 1795.521,A 0.000,B 0.000,C 90.000,E1 273.898} C_DIS
LIN {X -0.151,Y -337.129,Z 1795.519,A 0.000,B 0.000,C 90.000,E1 273.383} C_DIS
LIN {X 0.067,Y -330.841,Z 1795.516,A 0.000,B 0.000,C 90.000,E1 272.865} C_DIS
LIN {X -0.147,Y -324.418,Z 1795.514,A 0.000,B 0.000,C 90.000,E1 272.465} C_DIS
LIN {X -0.122,Y -317.836,Z 1795.511,A 0.000,B 0.000,C 90.000,E1 272.064} C_DIS
LIN {X 0.133,Y -310.692,Z 1795.509,A 0.000,B 0.000,C 90.000,E1 271.661} C_DIS
LIN {X 0.097,Y -303.502,Z 1795.508,A 0.000,B 0.000,C 90.000,E1 271.375} C_DIS
LIN {X 0.039,Y -295.840,Z 1795.506,A 0.000,B 0.000,C 90.000,E1 271.146} C_DIS
LIN {X 0.010,Y -281.206,Z 1795.505,A 0.000,B 0.000,C 90.000,E1 270.802} C_DIS
LIN {X 0.041,Y -265.842,Z 1795.503,A 0.000,B 0.000,C 90.000,E1 270.516} C_DIS
LIN {X -0.032,Y -253.378,Z 1795.502,A 0.000,B 0.000,C 90.000,E1 270.344} C_DIS
LIN {X -0.005,Y -239.249,Z 1795.501,A 0.000,B 0.000,C 90.000,E1 270.229} C_DIS
LIN {X -0.100,Y -232.241,Z 1795.501,A 0.000,B 0.000,C 90.000,E1 270.229} C_DIS
LIN {X 0.085,Y -181.580,Z 1795.501,A 0.000,B 0.000,C 90.000,E1 270.172} C_DIS
LIN {X 0.040,Y -180.802,Z 1795.471,A 0.000,B 0.000,C 90.000,E1 264.780} C_DIS
LIN {X -0.063,Y -178.902,Z 1795.443,A 0.000,B 0.000,C 90.000,E1 259.746} C_DIS
LIN {X 0.017,Y -175.946,Z 1795.415,A 0.000,B 0.000,C 90.000,E1 254.629} C_DIS
LIN {X -0.035,Y -175.406,Z 1795.410,A 0.000,B 0.000,C 90.000,E1 253.795} C_DIS
LIN {X -0.032,Y -172.172,Z 1795.386,A 0.000,B 0.000,C 90.000,E1 249.518} C_DIS
LIN {X 0.006,Y -171.642,Z 1795.381,A 0.000,B 0.000,C 90.000,E1 248.646} C_DIS
LIN {X 0.002,Y -167.865,Z 1795.357,A 0.000,B 0.000,C 90.000,E1 244.332} C_DIS
LIN {X -0.056,Y -166.598,Z 1795.348,A 0.000,B 0.000,C 90.000,E1 242.615} C_DIS
LIN {X 0.077,Y -162.587,Z 1795.323,A 0.000,B 0.000,C 90.000,E1 238.201} C_DIS
LIN {X -0.086,Y -161.271,Z 1795.314,A 0.000,B 0.000,C 90.000,E1 236.501} C_DIS
LIN {X -0.051,Y -157.272,Z 1795.289,A 0.000,B 0.000,C 90.000,E1 232.065} C_DIS
LIN {X -0.028,Y -155.990,Z 1795.279,A 0.000,B 0.000,C 90.000,E1 230.275} C_DIS
LIN {X -0.067,Y -152.248,Z 1795.254,A 0.000,B 0.000,C 90.000,E1 225.810} C_DIS
LIN {X -0.045,Y -150.488,Z 1795.239,A 0.000,B 0.000,C 90.000,E1 223.095} C_DIS
LIN {X -0.014,Y -147.212,Z 1795.214,A 0.000,B 0.000,C 90.000,E1 218.543} C_DIS
LIN {X -0.044,Y -145.233,Z 1795.194,A 0.000,B 0.000,C 90.000,E1 214.898} C_DIS
LIN {X 0.067,Y -142.356,Z 1795.163,A 0.000,B 0.000,C 90.000,E1 209.333} C_DIS
LIN {X -0.006,Y -141.744,Z 1795.153,A 0.000,B 0.000,C 90.000,E1 207.513} C_DIS
LIN {X -0.080,Y -139.489,Z 1795.117,A 0.000,B 0.000,C 90.000,E1 201.046} C_DIS
LIN {X -0.043,Y -138.992,Z 1795.101,A 0.000,B 0.000,C 90.000,E1 198.236} C_DIS
LIN {X 0.050,Y -138.336,Z 1795.055,A 0.000,B 0.000,C 90.000,E1 189.792} C_DIS
LIN {X -0.064,Y -139.418,Z 1795.008,A 0.000,B 0.000,C 90.000,E1 181.432} C_DIS
LIN {X -0.011,Y -141.335,Z 1794.972,A 0.000,B 0.000,C 90.000,E1 174.894} C_DIS
LIN {X -0.054,Y -142.691,Z 1794.956,A 0.000,B 0.000,C 90.000,E1 172.129} C_DIS
LIN {X 0.067,Y -145.054,Z 1794.931,A 0.000,B 0.000,C 90.000,E1 167.465} C_DIS
LIN {X 0.064,Y -147.680,Z 1794.910,A 0.000,B 0.000,C 90.000,E1 163.795} C_DIS
LIN {X -0.044,Y -150.325,Z 1794.890,A 0.000,B 0.000,C 90.000,E1 160.188} C_DIS
LIN {X 0.028,Y -153.741,Z 1794.870,A 0.000,B 0.000,C 90.000,E1 156.538} C_DIS
LIN {X 0.019,Y -157.155,Z 1794.850,A 0.000,B 0.000,C 90.000,E1 152.948} C_DIS
LIN {X -0.047,Y -161.305,Z 1794.830,A 0.000,B 0.000,C 90.000,E1 149.410} C_DIS
LIN {X -0.030,Y -164.420,Z 1794.815,A 0.000,B 0.000,C 90.000,E1 146.755} C_DIS
LIN {X -0.034,Y -169.104,Z 1794.796,A 0.000,B 0.000,C 90.000,E1 143.256} C_DIS
LIN {X -0.084,Y -171.659,Z 1794.786,A 0.000,B 0.000,C 90.000,E1 141.537} C_DIS
LIN {X -0.038,Y -176.624,Z 1794.767,A 0.000,B 0.000,C 90.000,E1 138.081} C_DIS
LIN {X 0.091,Y -180.922,Z 1794.753,A 0.000,B 0.000,C 90.000,E1 135.486} C_DIS
LIN {X -0.046,Y -186.341,Z 1794.734,A 0.000,B 0.000,C 90.000,E1 132.162} C_DIS
LIN {X 0.021,Y -190.973,Z 1794.720,A 0.000,B 0.000,C 90.000,E1 129.644} C_DIS
LIN {X -0.061,Y -196.747,Z 1794.702,A 0.000,B 0.000,C 90.000,E1 126.377} C_DIS
LIN {X -0.029,Y -199.995,Z 1794.693,A 0.000,B 0.000,C 90.000,E1 124.739} C_DIS
LIN {X -0.048,Y -207.498,Z 1794.671,A 0.000,B 0.000,C 90.000,E1 120.718} C_DIS
LIN {X 0.022,Y -211.121,Z 1794.660,A 0.000,B 0.000,C 90.000,E1 118.871} C_DIS
LIN {X -0.034,Y -211.952,Z 1794.658,A 0.000,B 0.000,C 90.000,E1 118.409} C_DIS
LIN {X -0.089,Y -338.288,Z 1794.658,A 0.000,B 0.000,C 90.000,E1 118.409} C_DIS
LIN {X 0.081,Y -341.237,Z 1794.657,A 0.000,B 0.000,C 90.000,E1 118.309} C_DIS
LIN {X -0.014,Y -344.255,Z 1794.656,A 0.000,B 0.000,C 90.000,E1 118.153} C_DIS
LIN {X -0.074,Y -347.689,Z 1794.655,A 0.000,B 0.000,C 90.000,E1 117.820} C_DIS
LIN {X 0.021,Y -350.870,Z 1794.651,A 0.000,B 0.000,C 90.000,E1 117.257} C_DIS
LIN {X -0.026,Y -360.196,Z 1794.638,A 0.000,B 0.000,C 90.000,E1 114.847} C_DIS
LIN {X -0.143,Y -367.115,Z 1794.628,A 0.000,B 0.000,C 90.000,E1 113.078} C_DIS
LIN {X -0.044,Y -372.566,Z 1794.620,A 0.000,B 0.000,C 90.000,E1 111.589} C_DIS
LIN {X -0.222,Y -375.481,Z 1794.615,A 0.000,B 0.000,C 90.000,E1 110.737} C_DIS
LIN {X -0.006,Y -377.121,Z 1794.612,A 0.000,B 0.000,C 90.000,E1 110.120} C_DIS
LIN {X 0.093,Y -378.287,Z 1794.609,A 0.000,B 0.000,C 90.000,E1 109.523} C_DIS
LIN {X -0.029,Y -378.316,Z 1794.605,A 0.000,B 0.000,C 90.000,E1 108.960} C_DIS
LIN {X 0.000,Y -371.626,Z 1794.576,A 0.000,B 0.000,C 90.000,E1 103.716} C_DIS
LIN {X -0.076,Y -369.302,Z 1794.559,A 0.000,B 0.000,C 90.000,E1 100.658} C_DIS
LIN {X -0.135,Y -369.387,Z 1794.559,A 0.000,B 0.000,C 90.000,E1 100.658} C_DIS
LIN {X 0.096,Y -387.072,Z 1794.549,A 0.000,B 0.000,C 90.000,E1 98.859} C_DIS
LIN {X -0.152,Y -406.265,Z 1794.540,A 0.000,B 0.000,C 90.000,E1 97.182} C_DIS
LIN {X -0.034,Y -428.587,Z 1794.530,A 0.000,B 0.000,C 90.000,E1 95.391} C_DIS
LIN {X -0.169,Y -439.698,Z 1794.525,A 0.000,B 0.000,C 90.000,E1 94.588} C_DIS
LIN {X 0.106,Y -443.387,Z 1794.523,A 0.000,B 0.000,C 90.000,E1 94.131} C_DIS
LIN {X -0.140,Y -444.954,Z 1794.522,A 0.000,B 0.000,C 90.000,E1 93.898} C_DIS
LIN {X 0.028,Y -446.134,Z 1794.520,A 0.000,B 0.000,C 90.000,E1 93.612} C_DIS
LIN {X -0.022,Y -447.583,Z 1794.517,A 0.000,B 0.000,C 90.000,E1 93.094} C_DIS
LIN {X -0.090,Y -448.034,Z 1794.514,A 0.000,B 0.000,C 90.000,E1 92.579} C_DIS
LIN {X -0.147,Y -447.559,Z 1794.511,A 0.000,B 0.000,C 90.000,E1 92.064} C_DIS
LIN {X -0.185,Y -446.092,Z 1794.508,A 0.000,B 0.000,C 90.000,E1 91.547} C_DIS
LIN {X 0.010,Y -444.912,Z 1794.507,A 0.000,B 0.000,C 90.000,E1 91.260} C_DIS
LIN {X 0.047,Y -436.738,Z 1794.500,A 0.000,B 0.000,C 90.000,E1 89.943} C_DIS
LIN {X 0.104,Y -426.846,Z 1794.491,A 0.000,B 0.000,C 90.000,E1 88.339} C_DIS
LIN {X 0.115,Y -415.074,Z 1794.480,A 0.000,B 0.000,C 90.000,E1 86.445} C_DIS
LIN {X -0.167,Y -404.922,Z 1794.471,A 0.000,B 0.000,C 90.000,E1 84.837} C_DIS
LIN {X -0.113,Y -392.990,Z 1794.460,A 0.000,B 0.000,C 90.000,E1 82.875} C_DIS
LIN {X 0.164,Y -381.411,Z 1794.450,A 0.000,B 0.000,C 90.000,E1 80.905} C_DIS
LIN {X 0.104,Y -381.409,Z 1794.450,A 0.000,B 0.000,C 90.000,E1 80.905} C_DIS
LIN {X -0.185,Y -384.343,Z 1794.441,A 0.000,B 0.000,C 90.000,E1 79.454} C_DIS
LIN {X -0.125,Y -385.305,Z 1794.438,A 0.000,B 0.000,C 90.000,E1 78.870} C_DIS
LIN {X -0.056,Y -384.865,Z 1794.435,A 0.000,B 0.000,C 90.000,E1 78.285} C_DIS
LIN {X 0.017,Y -383.770,Z 1794.432,A 0.000,B 0.000,C 90.000,E1 77.701} C_DIS
LIN {X 0.086,Y -382.349,Z 1794.428,A 0.000,B 0.000,C 90.000,E1 77.117} C_DIS
LIN {X -0.083,Y -378.957,Z 1794.422,A 0.000,B 0.000,C 90.000,E1 75.992} C_DIS
LIN {X 0.190,Y -373.143,Z 1794.412,A 0.000,B 0.000,C 90.000,E1 74.212} C_DIS
LIN {X -0.008,Y -366.895,Z 1794.403,A 0.000,B 0.000,C 90.000,E1 72.489} C_DIS
LIN {X -0.097,Y -360.348,Z 1794.393,A 0.000,B 0.000,C 90.000,E1 70.732} C_DIS
LIN {X 0.180,Y -352.466,Z 1794.381,A 0.000,B 0.000,C 90.000,E1 68.592} C_DIS
LIN {X 0.066,Y -345.608,Z 1794.371,A 0.000,B 0.000,C 90.000,E1 66.794} C_DIS
LIN {X -0.034,Y -337.467,Z 1794.359,A 0.000,B 0.000,C 90.000,E1 64.665} C_DIS
LIN {X 0.009,Y -330.297,Z 1794.349,A 0.000,B 0.000,C 90.000,E1 62.794} C_DIS
LIN {X -0.179,Y -323.913,Z 1794.340,A 0.000,B 0.000,C 90.000,E1 61.257} C_DIS
LIN {X -0.152,Y -316.993,Z 1794.331,A 0.000,B 0.000,C 90.000,E1 59.665} C_DIS
LIN {X -0.070,Y -309.609,Z 1794.322,A 0.000,B 0.000,C 90.000,E1 58.043} C_DIS
LIN {X -0.072,Y -300.626,Z 1794.312,A 0.000,B 0.000,C 90.000,E1 56.087} C_DIS
LIN {X 0.010,Y -290.207,Z 1794.299,A 0.000,B 0.000,C 90.000,E1 53.749} C_DIS
LIN {X -0.001,Y -275.885,Z 1794.280,A 0.000,B 0.000,C 90.000,E1 50.356} C_DIS
LIN {X -0.033,Y -264.004,Z 1794.262,A 0.000,B 0.000,C 90.000,E1 47.229} C_DIS
LIN {X -0.043,Y -252.763,Z 1794.245,A 0.000,B 0.000,C 90.000,E1 44.028} C_DIS
LIN {X -0.160,Y -243.286,Z 1794.228,A 0.000,B 0.000,C 90.000,E1 41.148} C_DIS
LIN {X -0.117,Y -234.151,Z 1794.212,A 0.000,B 0.000,C 90.000,E1 38.177} C_DIS
LIN {X 0.114,Y -225.479,Z 1794.195,A 0.000,B 0.000,C 90.000,E1 35.105} C_DIS
LIN {X -0.059,Y -217.338,Z 1794.178,A 0.000,B 0.000,C 90.000,E1 32.084} C_DIS
LIN {X 0.009,Y -209.769,Z 1794.161,A 0.000,B 0.000,C 90.000,E1 28.949} C_DIS
LIN {X -0.045,Y -202.882,Z 1794.143,A 0.000,B 0.000,C 90.000,E1 25.796} C_DIS
LIN {X -0.071,Y -196.808,Z 1794.125,A 0.000,B 0.000,C 90.000,E1 22.589} C_DIS
LIN {X -0.040,Y -191.581,Z 1794.107,A 0.000,B 0.000,C 90.000,E1 19.322} C_DIS
LIN {X -0.028,Y -187.299,Z 1794.089,A 0.000,B 0.000,C 90.000,E1 16.024} C_DIS
LIN {X 0.086,Y -183.125,Z 1794.066,A 0.000,B 0.000,C 90.000,E1 11.827} C_DIS
LIN {X 0.031,Y -179.975,Z 1794.042,A 0.000,B 0.000,C 90.000,E1 7.644} C_DIS
LIN {X 0.032,Y -177.378,Z 1794.010,A 0.000,B 0.000,C 90.000,E1 1.718} C_DIS
LIN {X -0.068,Y -176.464,Z 1793.974,A 0.000,B 0.000,C 90.000,E1 355.298} C_DIS
LIN {X -0.001,Y -177.281,Z 1793.936,A 0.000,B 0.000,C 90.000,E1 348.465} C_DIS
LIN {X -0.066,Y -179.402,Z 1793.903,A 0.000,B 0.000,C 90.000,E1 342.543} C_DIS
LIN {X -0.099,Y -182.355,Z 1793.875,A 0.000,B 0.000,C 90.000,E1 337.486} C_DIS
LIN {X 0.047,Y -186.170,Z 1793.847,A 0.000,B 0.000,C 90.000,E1 332.410} C_DIS
LIN {X -0.043,Y -190.070,Z 1793.824,A 0.000,B 0.000,C 90.000,E1 328.280} C_DIS
LIN {X -0.006,Y -194.928,Z 1793.801,A 0.000,B 0.000,C 90.000,E1 324.149} C_DIS
LIN {X 0.006,Y -199.806,Z 1793.783,A 0.000,B 0.000,C 90.000,E1 320.884} C_DIS
LIN {X 0.092,Y -205.891,Z 1793.765,A 0.000,B 0.000,C 90.000,E1 317.634} C_DIS
LIN {X 0.092,Y -211.350,Z 1793.751,A 0.000,B 0.000,C 90.000,E1 315.243} C_DIS
LIN {X 0.004,Y -216.681,Z 1793.741,A 0.000,B 0.000,C 90.000,E1 313.299} C_DIS
LIN {X -0.059,Y -221.584,Z 1793.732,A 0.000,B 0.000,C 90.000,E1 311.757} C_DIS
LIN {X 0.112,Y -227.220,Z 1793.723,A 0.000,B 0.000,C 90.000,E1 310.172} C_DIS
LIN {X -0.014,Y -235.240,Z 1793.713,A 0.000,B 0.000,C 90.000,E1 308.302} C_DIS
LIN {X 0.026,Y -244.346,Z 1793.702,A 0.000,B 0.000,C 90.000,E1 306.423} C_DIS
LIN {X -0.066,Y -256.505,Z 1793.690,A 0.000,B 0.000,C 90.000,E1 304.246} C_DIS
LIN {X -0.015,Y -274.439,Z 1793.674,A 0.000,B 0.000,C 90.000,E1 301.386} C_DIS
LIN {X 0.111,Y -291.439,Z 1793.661,A 0.000,B 0.000,C 90.000,E1 298.949} C_DIS
LIN {X -0.012,Y -311.911,Z 1793.646,A 0.000,B 0.000,C 90.000,E1 296.309} C_DIS
LIN {X -0.021,Y -325.054,Z 1793.637,A 0.000,B 0.000,C 90.000,E1 294.695} C_DIS
LIN {X -0.083,Y -335.430,Z 1793.630,A 0.000,B 0.000,C 90.000,E1 293.439} C_DIS
LIN {X -0.103,Y -347.962,Z 1793.622,A 0.000,B 0.000,C 90.000,E1 291.897} C_DIS
LIN {X -0.007,Y -357.650,Z 1793.615,A 0.000,B 0.000,C 90.000,E1 290.663} C_DIS
LIN {X 0.025,Y -364.423,Z 1793.610,A 0.000,B 0.000,C 90.000,E1 289.758} C_DIS
LIN {X 0.121,Y -370.655,Z 1793.605,A 0.000,B 0.000,C 90.000,E1 288.852} C_DIS
LIN {X -0.071,Y -375.997,Z 1793.600,A 0.000,B 0.000,C 90.000,E1 288.000} C_DIS
LIN {X 0.025,Y -379.058,Z 1793.597,A 0.000,B 0.000,C 90.000,E1 287.402} C_DIS
LIN {X 0.144,Y -381.665,Z 1793.594,A 0.000,B 0.000,C 90.000,E1 286.804} C_DIS
LIN {X -0.068,Y -384.867,Z 1793.589,A 0.000,B 0.000,C 90.000,E1 285.969} C_DIS
LIN {X 0.091,Y -386.531,Z 1793.585,A 0.000,B 0.000,C 90.000,E1 285.371} C_DIS
LIN {X -0.120,Y -387.853,Z 1793.582,A 0.000,B 0.000,C 90.000,E1 284.828} C_DIS
LIN {X -0.046,Y -388.823,Z 1793.579,A 0.000,B 0.000,C 90.000,E1 284.245} C_DIS
LIN {X 0.133,Y -389.406,Z 1793.576,A 0.000,B 0.000,C 90.000,E1 283.647} C_DIS
LIN {X -0.153,Y -389.644,Z 1793.573,A 0.000,B 0.000,C 90.000,E1 283.119} C_DIS
LIN {X -0.056,Y -389.503,Z 1793.570,A 0.000,B 0.000,C 90.000,E1 282.535} C_DIS
LIN {X 0.045,Y -388.982,Z 1793.566,A 0.000,B 0.000,C 90.000,E1 281.951} C_DIS
LIN {X 0.145,Y -388.126,Z 1793.563,A 0.000,B 0.000,C 90.000,E1 281.366} C_DIS
LIN {X -0.138,Y -386.913,Z 1793.560,A 0.000,B 0.000,C 90.000,E1 280.838} C_DIS
LIN {X -0.048,Y -385.339,Z 1793.557,A 0.000,B 0.000,C 90.000,E1 280.254} C_DIS
LIN {X 0.068,Y -382.300,Z 1793.552,A 0.000,B 0.000,C 90.000,E1 279.378} C_DIS
LIN {X 0.092,Y -378.686,Z 1793.547,A 0.000,B 0.000,C 90.000,E1 278.511} C_DIS
LIN {X 0.082,Y -374.206,Z 1793.542,A 0.000,B 0.000,C 90.000,E1 277.644} C_DIS
LIN {X 0.036,Y -368.850,Z 1793.538,A 0.000,B 0.000,C 90.000,E1 276.777} C_DIS
LIN {X -0.061,Y -362.514,Z 1793.533,A 0.000,B 0.000,C 90.000,E1 275.910} C_DIS
LIN {X -0.167,Y -357.602,Z 1793.530,A 0.000,B 0.000,C 90.000,E1 275.334} C_DIS
LIN {X 0.118,Y -352.138,Z 1793.526,A 0.000,B 0.000,C 90.000,E1 274.702} C_DIS
LIN {X 0.160,Y -346.434,Z 1793.523,A 0.000,B 0.000,C 90.000,E1 274.131} C_DIS
LIN {X 0.083,Y -340.517,Z 1793.520,A 0.000,B 0.000,C 90.000,E1 273.612} C_DIS
LIN {X -0.116,Y -334.426,Z 1793.517,A 0.000,B 0.000,C 90.000,E1 273.151} C_DIS
LIN {X -0.107,Y -328.120,Z 1793.515,A 0.000,B 0.000,C 90.000,E1 272.694} C_DIS
LIN {X 0.127,Y -321.668,Z 1793.513,A 0.000,B 0.000,C 90.000,E1 272.236} C_DIS
LIN {X -0.056,Y -314.916,Z 1793.510,A 0.000,B 0.000,C 90.000,E1 271.892} C_DIS
LIN {X 0.050,Y -307.801,Z 1793.509,A 0.000,B 0.000,C 90.000,E1 271.547} C_DIS
LIN {X -0.148,Y -300.326,Z 1793.507,A 0.000,B 0.000,C 90.000,E1 271.318} C_DIS
LIN {X 0.045,Y -288.908,Z 1793.505,A 0.000,B 0.000,C 90.000,E1 270.974} C_DIS
LIN {X 0.000,Y -278.155,Z 1793.504,A 0.000,B 0.000,C 90.000,E1 270.745} C_DIS
LIN {X 0.070,Y -262.412,Z 1793.503,A 0.000,B 0.000,C 90.000,E1 270.458} C_DIS
LIN {X 0.030,Y -253.803,Z 1793.502,A 0.000,B 0.000,C 90.000,E1 270.344} C_DIS
LIN {X 0.066,Y -240.225,Z 1793.501,A 0.000,B 0.000,C 90.000,E1 270.229} C_DIS
LIN {X -0.041,Y -232.821,Z 1793.501,A 0.000,B 0.000,C 90.000,E1 270.229} C_DIS
LIN {X -0.053,Y -181.580,Z 1793.501,A 0.000,B 0.000,C 90.000,E1 270.229} C_DIS
LIN {X 0.076,Y -180.806,Z 1793.471,A 0.000,B 0.000,C 90.000,E1 264.780} C_DIS
LIN {X -0.026,Y -178.907,Z 1793.443,A 0.000,B 0.000,C 90.000,E1 259.746} C_DIS
LIN {X 0.054,Y -175.951,Z 1793.415,A 0.000,B 0.000,C 90.000,E1 254.629} C_DIS
LIN {X 0.001,Y -175.416,Z 1793.410,A 0.000,B 0.000,C 90.000,E1 253.795} C_DIS
LIN {X 0.004,Y -172.179,Z 1793.386,A 0.000,B 0.000,C 90.000,E1 249.518} C_DIS
LIN {X 0.043,Y -171.650,Z 1793.381,A 0.000,B 0.000,C 90.000,E1 248.646} C_DIS
LIN {X 0.037,Y -167.874,Z 1793.357,A 0.000,B 0.000,C 90.000,E1 244.332} C_DIS
LIN {X -0.020,Y -166.609,Z 1793.348,A 0.000,B 0.000,C 90.000,E1 242.615} C_DIS
LIN {X -0.026,Y -162.597,Z 1793.324,A 0.000,B 0.000,C 90.000,E1 238.250} C_DIS
LIN {X -0.052,Y -161.282,Z 1793.314,A 0.000,B 0.000,C 90.000,E1 236.501} C_DIS
LIN {X -0.017,Y -157.281,Z 1793.289,A 0.000,B 0.000,C 90.000,E1 232.065} C_DIS
LIN {X 0.006,Y -155.999,Z 1793.279,A 0.000,B 0.000,C 90.000,E1 230.275} C_DIS
LIN {X -0.033,Y -152.256,Z 1793.254,A 0.000,B 0.000,C 90.000,E1 225.810} C_DIS
LIN {X -0.011,Y -150.496,Z 1793.239,A 0.000,B 0.000,C 90.000,E1 223.095} C_DIS
LIN {X 0.019,Y -147.220,Z 1793.214,A 0.000,B 0.000,C 90.000,E1 218.543} C_DIS
LIN {X -0.011,Y -145.241,Z 1793.194,A 0.000,B 0.000,C 90.000,E1 214.898} C_DIS
LIN {X 0.030,Y -142.361,Z 1793.163,A 0.000,B 0.000,C 90.000,E1 209.361} C_DIS
LIN {X 0.026,Y -141.748,Z 1793.153,A 0.000,B 0.000,C 90.000,E1 207.513} C_DIS
LIN {X -0.048,Y -139.492,Z 1793.117,A 0.000,B 0.000,C 90.000,E1 201.046} C_DIS
LIN {X -0.011,Y -138.995,Z 1793.101,A 0.000,B 0.000,C 90.000,E1 198.236} C_DIS
LIN {X -0.054,Y -138.336,Z 1793.055,A 0.000,B 0.000,C 90.000,E1 189.849} C_DIS
LIN {X -0.032,Y -139.415,Z 1793.008,A 0.000,B 0.000,C 90.000,E1 181.432} C_DIS
LIN {X 0.021,Y -141.329,Z 1792.972,A 0.000,B 0.000,C 90.000,E1 174.894} C_DIS
LIN {X -0.021,Y -142.686,Z 1792.956,A 0.000,B 0.000,C 90.000,E1 172.129} C_DIS
LIN {X -0.042,Y -145.046,Z 1792.931,A 0.000,B 0.000,C 90.000,E1 167.521} C_DIS
LIN {X -0.045,Y -147.672,Z 1792.910,A 0.000,B 0.000,C 90.000,E1 163.850} C_DIS
LIN {X -0.010,Y -150.314,Z 1792.890,A 0.000,B 0.000,C 90.000,E1 160.188} C_DIS
LIN {X 0.062,Y -153.728,Z 1792.870,A 0.000,B 0.000,C 90.000,E1 156.538} C_DIS
LIN {X -0.086,Y -157.141,Z 1792.850,A 0.000,B 0.000,C 90.000,E1 152.999} C_DIS
LIN {X -0.012,Y -161.289,Z 1792.830,A 0.000,B 0.000,C 90.000,E1 149.410} C_DIS
LIN {X 0.005,Y -164.406,Z 1792.815,A 0.000,B 0.000,C 90.000,E1 146.755} C_DIS
LIN {X 0.003,Y -169.087,Z 1792.796,A 0.000,B 0.000,C 90.000,E1 143.256} C_DIS
LIN {X -0.046,Y -171.644,Z 1792.786,A 0.000,B 0.000,C 90.000,E1 141.537} C_DIS
LIN {X 0.000,Y -176.606,Z 1792.767,A 0.000,B 0.000,C 90.000,E1 138.081} C_DIS
LIN {X 0.001,Y -180.904,Z 1792.753,A 0.000,B 0.000,C 90.000,E1 135.526} C_DIS
LIN {X -0.007,Y -186.320,Z 1792.734,A 0.000,B 0.000,C 90.000,E1 132.162} C_DIS
LIN {X 0.059,Y -190.954,Z 1792.720,A 0.000,B 0.000,C 90.000,E1 129.644} C_DIS
LIN {X -0.021,Y -196.725,Z 1792.702,A 0.000,B 0.000,C 90.000,E1 126.377} C_DIS
LIN {X 0.010,Y -199.972,Z 1792.693,A 0.000,B 0.000,C 90.000,E1 124.739} C_DIS
LIN {X -0.007,Y -207.475,Z 1792.671,A 0.000,B 0.000,C 90.000,E1 120.718} C_DIS
LIN {X 0.057,Y -211.191,Z 1792.660,A 0.000,B 0.000,C 90.000,E1 118.821} C_DIS
LIN {X 0.065,Y -211.632,Z 1792.659,A 0.000,B 0.000,C 90.000,E1 118.565} C_DIS
LIN {X 0.063,Y -338.331,Z 1792.659,A 0.000,B 0.000,C 90.000,E1 118.565} C_DIS
LIN {X -0.155,Y -344.456,Z 1792.657,A 0.000,B 0.000,C 90.000,E1 118.359} C_DIS
LIN {X -0.098,Y -347.210,Z 1792.656,A 0.000,B 0.000,C 90.000,E1 118.103} C_DIS
LIN {X -0.045,Y -350.725,Z 1792.653,A 0.000,B 0.000,C 90.000,E1 117.590} C_DIS
LIN {X -0.169,Y -353.357,Z 1792.650,A 0.000,B 0.000,C 90.000,E1 117.001} C_DIS
LIN {X 0.076,Y -364.476,Z 1792.635,A 0.000,B 0.000,C 90.000,E1 114.259} C_DIS
LIN {X -0.022,Y -373.218,Z 1792.623,A 0.000,B 0.000,C 90.000,E1 112.206} C_DIS
LIN {X 0.038,Y -379.260,Z 1792.615,A 0.000,B 0.000,C 90.000,E1 110.737} C_DIS
LIN {X 0.056,Y -383.698,Z 1792.609,A 0.000,B 0.000,C 90.000,E1 109.577} C_DIS
LIN {X -0.021,Y -386.493,Z 1792.604,A 0.000,B 0.000,C 90.000,E1 108.725} C_DIS
LIN {X 0.142,Y -387.805,Z 1792.601,A 0.000,B 0.000,C 90.000,E1 108.127} C_DIS
LIN {X -0.052,Y -387.975,Z 1792.598,A 0.000,B 0.000,C 90.000,E1 107.583} C_DIS
LIN {X 0.098,Y -381.649,Z 1792.566,A 0.000,B 0.000,C 90.000,E1 101.827} C_DIS
LIN {X -0.150,Y -380.278,Z 1792.553,A 0.000,B 0.000,C 90.000,E1 99.557} C_DIS
LIN {X 0.165,Y -380.311,Z 1792.553,A 0.000,B 0.000,C 90.000,E1 99.500} C_DIS
LIN {X 0.088,Y -399.832,Z 1792.543,A 0.000,B 0.000,C 90.000,E1 97.701} C_DIS
LIN {X -0.182,Y -422.034,Z 1792.533,A 0.000,B 0.000,C 90.000,E1 95.910} C_DIS
LIN {X -0.095,Y -438.897,Z 1792.526,A 0.000,B 0.000,C 90.000,E1 94.645} C_DIS
LIN {X 0.115,Y -441.080,Z 1792.525,A 0.000,B 0.000,C 90.000,E1 94.416} C_DIS
LIN {X 0.023,Y -443.055,Z 1792.523,A 0.000,B 0.000,C 90.000,E1 94.188} C_DIS
LIN {X -0.037,Y -444.569,Z 1792.522,A 0.000,B 0.000,C 90.000,E1 93.955} C_DIS
LIN {X 0.140,Y -445.836,Z 1792.521,A 0.000,B 0.000,C 90.000,E1 93.669} C_DIS
LIN {X -0.126,Y -446.777,Z 1792.519,A 0.000,B 0.000,C 90.000,E1 93.440} C_DIS
LIN {X -0.171,Y -447.842,Z 1792.516,A 0.000,B 0.000,C 90.000,E1 92.922} C_DIS
LIN {X 0.213,Y -447.954,Z 1792.513,A 0.000,B 0.000,C 90.000,E1 92.350} C_DIS
LIN {X 0.159,Y -447.132,Z 1792.510,A 0.000,B 0.000,C 90.000,E1 91.835} C_DIS
LIN {X 0.118,Y -445.249,Z 1792.507,A 0.000,B 0.000,C 90.000,E1 91.318} C_DIS
LIN {X 0.061,Y -442.147,Z 1792.505,A 0.000,B 0.000,C 90.000,E1 90.802} C_DIS
LIN {X 0.082,Y -428.941,Z 1792.493,A 0.000,B 0.000,C 90.000,E1 88.682} C_DIS
LIN {X 0.011,Y -418.886,Z 1792.484,A 0.000,B 0.000,C 90.000,E1 87.078} C_DIS
LIN {X -0.207,Y -408.759,Z 1792.475,A 0.000,B 0.000,C 90.000,E1 85.469} C_DIS
LIN {X -0.123,Y -396.870,Z 1792.464,A 0.000,B 0.000,C 90.000,E1 83.514} C_DIS
LIN {X -0.075,Y -390.548,Z 1792.458,A 0.000,B 0.000,C 90.000,E1 82.470} C_DIS
LIN {X -0.137,Y -390.544,Z 1792.458,A 0.000,B 0.000,C 90.000,E1 82.470} C_DIS
LIN {X -0.141,Y -393.247,Z 1792.450,A 0.000,B 0.000,C 90.000,E1 80.971} C_DIS
LIN {X -0.028,Y -394.113,Z 1792.447,A 0.000,B 0.000,C 90.000,E1 80.387} C_DIS
LIN {X 0.094,Y -393.600,Z 1792.443,A 0.000,B 0.000,C 90.000,E1 79.803} C_DIS
LIN {X 0.223,Y -392.432,Z 1792.440,A 0.000,B 0.000,C 90.000,E1 79.218} C_DIS
LIN {X -0.113,Y -390.924,Z 1792.437,A 0.000,B 0.000,C 90.000,E1 78.701} C_DIS
LIN {X 0.191,Y -387.347,Z 1792.431,A 0.000,B 0.000,C 90.000,E1 77.521} C_DIS
LIN {X -0.005,Y -383.368,Z 1792.424,A 0.000,B 0.000,C 90.000,E1 76.408} C_DIS
LIN {X -0.017,Y -376.952,Z 1792.415,A 0.000,B 0.000,C 90.000,E1 74.685} C_DIS
LIN {X -0.146,Y -370.287,Z 1792.405,A 0.000,B 0.000,C 90.000,E1 72.960} C_DIS
LIN {X 0.158,Y -363.439,Z 1792.395,A 0.000,B 0.000,C 90.000,E1 71.148} C_DIS
LIN {X 0.043,Y -355.210,Z 1792.384,A 0.000,B 0.000,C 90.000,E1 69.082} C_DIS
LIN {X 0.013,Y -346.918,Z 1792.372,A 0.000,B 0.000,C 90.000,E1 66.975} C_DIS
LIN {X -0.059,Y -338.482,Z 1792.360,A 0.000,B 0.000,C 90.000,E1 64.845} C_DIS
LIN {X -0.143,Y -331.102,Z 1792.350,A 0.000,B 0.000,C 90.000,E1 62.999} C_DIS
LIN {X 0.124,Y -324.575,Z 1792.341,A 0.000,B 0.000,C 90.000,E1 61.385} C_DIS
LIN {X 0.152,Y -317.495,Z 1792.332,A 0.000,B 0.000,C 90.000,E1 59.793} C_DIS
LIN {X 0.076,Y -310.146,Z 1792.323,A 0.000,B 0.000,C 90.000,E1 58.201} C_DIS
LIN {X -0.177,Y -301.167,Z 1792.313,A 0.000,B 0.000,C 90.000,E1 56.294} C_DIS
LIN {X 0.152,Y -290.681,Z 1792.300,A 0.000,B 0.000,C 90.000,E1 53.909} C_DIS
LIN {X -0.071,Y -276.349,Z 1792.281,A 0.000,B 0.000,C 90.000,E1 50.561} C_DIS
LIN {X 0.118,Y -264.395,Z 1792.263,A 0.000,B 0.000,C 90.000,E1 47.391} C_DIS
LIN {X -0.050,Y -251.890,Z 1792.244,A 0.000,B 0.000,C 90.000,E1 43.866} C_DIS
LIN {X -0.006,Y -242.399,Z 1792.227,A 0.000,B 0.000,C 90.000,E1 40.943} C_DIS
LIN {X 0.014,Y -233.290,Z 1792.211,A 0.000,B 0.000,C 90.000,E1 37.971} C_DIS
LIN {X 0.037,Y -224.615,Z 1792.194,A 0.000,B 0.000,C 90.000,E1 34.945} C_DIS
LIN {X 0.024,Y -216.514,Z 1792.177,A 0.000,B 0.000,C 90.000,E1 31.878} C_DIS
LIN {X 0.066,Y -208.971,Z 1792.160,A 0.000,B 0.000,C 90.000,E1 28.743} C_DIS
LIN {X -0.013,Y -202.111,Z 1792.142,A 0.000,B 0.000,C 90.000,E1 25.591} C_DIS
LIN {X -0.066,Y -196.098,Z 1792.124,A 0.000,B 0.000,C 90.000,E1 22.386} C_DIS
LIN {X 0.057,Y -190.911,Z 1792.106,A 0.000,B 0.000,C 90.000,E1 19.087} C_DIS
LIN {X 0.053,Y -186.689,Z 1792.088,A 0.000,B 0.000,C 90.000,E1 15.788} C_DIS
LIN {X -0.070,Y -182.570,Z 1792.065,A 0.000,B 0.000,C 90.000,E1 11.658} C_DIS
LIN {X 0.070,Y -179.481,Z 1792.041,A 0.000,B 0.000,C 90.000,E1 7.409} C_DIS
LIN {X 0.034,Y -176.959,Z 1792.008,A 0.000,B 0.000,C 90.000,E1 1.489} C_DIS
LIN {X -0.079,Y -176.127,Z 1791.974,A 0.000,B 0.000,C 90.000,E1 355.298} C_DIS
LIN {X -0.028,Y -176.960,Z 1791.936,A 0.000,B 0.000,C 90.000,E1 348.465} C_DIS
LIN {X 0.063,Y -179.075,Z 1791.903,A 0.000,B 0.000,C 90.000,E1 342.489} C_DIS
LIN {X 0.086,Y -182.065,Z 1791.875,A 0.000,B 0.000,C 90.000,E1 337.411} C_DIS
LIN {X -0.018,Y -185.904,Z 1791.847,A 0.000,B 0.000,C 90.000,E1 332.410} C_DIS
LIN {X -0.018,Y -189.864,Z 1791.824,A 0.000,B 0.000,C 90.000,E1 328.250} C_DIS
LIN {X 0.025,Y -194.813,Z 1791.801,A 0.000,B 0.000,C 90.000,E1 324.116} C_DIS
LIN {X -0.082,Y -199.763,Z 1791.783,A 0.000,B 0.000,C 90.000,E1 320.884} C_DIS
LIN {X 0.001,Y -205.945,Z 1791.765,A 0.000,B 0.000,C 90.000,E1 317.634} C_DIS
LIN {X -0.001,Y -211.468,Z 1791.751,A 0.000,B 0.000,C 90.000,E1 315.243} C_DIS
LIN {X -0.090,Y -216.831,Z 1791.740,A 0.000,B 0.000,C 90.000,E1 313.299} C_DIS
LIN {X 0.013,Y -221.774,Z 1791.732,A 0.000,B 0.000,C 90.000,E1 311.714} C_DIS
LIN {X 0.018,Y -227.420,Z 1791.723,A 0.000,B 0.000,C 90.000,E1 310.172} C_DIS
LIN {X 0.077,Y -235.478,Z 1791.713,A 0.000,B 0.000,C 90.000,E1 308.257} C_DIS
LIN {X -0.066,Y -244.631,Z 1791.702,A 0.000,B 0.000,C 90.000,E1 306.423} C_DIS
LIN {X 0.054,Y -256.817,Z 1791.690,A 0.000,B 0.000,C 90.000,E1 304.199} C_DIS
LIN {X 0.130,Y -274.806,Z 1791.674,A 0.000,B 0.000,C 90.000,E1 301.337} C_DIS
LIN {X 0.005,Y -294.334,Z 1791.659,A 0.000,B 0.000,C 90.000,E1 298.615} C_DIS
LIN {X -0.001,Y -314.922,Z 1791.644,A 0.000,B 0.000,C 90.000,E1 295.976} C_DIS
LIN {X -0.072,Y -330.601,Z 1791.634,A 0.000,B 0.000,C 90.000,E1 294.079} C_DIS
LIN {X 0.047,Y -343.172,Z 1791.625,A 0.000,B 0.000,C 90.000,E1 292.514} C_DIS
LIN {X 0.087,Y -353.111,Z 1791.618,A 0.000,B 0.000,C 90.000,E1 291.280} C_DIS
LIN {X 0.127,Y -362.501,Z 1791.612,A 0.000,B 0.000,C 90.000,E1 290.066} C_DIS
LIN {X -0.135,Y -368.939,Z 1791.607,A 0.000,B 0.000,C 90.000,E1 289.214} C_DIS
LIN {X 0.004,Y -374.643,Z 1791.602,A 0.000,B 0.000,C 90.000,E1 288.308} C_DIS
LIN {X -0.156,Y -379.411,Z 1791.597,A 0.000,B 0.000,C 90.000,E1 287.457} C_DIS
LIN {X 0.082,Y -383.161,Z 1791.592,A 0.000,B 0.000,C 90.000,E1 286.551} C_DIS
LIN {X 0.121,Y -385.221,Z 1791.589,A 0.000,B 0.000,C 90.000,E1 285.969} C_DIS
LIN {X -0.091,Y -386.893,Z 1791.586,A 0.000,B 0.000,C 90.000,E1 285.426} C_DIS
LIN {X 0.074,Y -388.234,Z 1791.582,A 0.000,B 0.000,C 90.000,E1 284.828} C_DIS
LIN {X 0.152,Y -389.191,Z 1791.579,A 0.000,B 0.000,C 90.000,E1 284.245} C_DIS
LIN {X -0.045,Y -389.781,Z 1791.576,A 0.000,B 0.000,C 90.000,E1 283.703} C_DIS
LIN {X 0.049,Y -390.011,Z 1791.573,A 0.000,B 0.000,C 90.000,E1 283.119} C_DIS
LIN {X 0.148,Y -389.910,Z 1791.570,A 0.000,B 0.000,C 90.000,E1 282.535} C_DIS
LIN {X -0.130,Y -389.413,Z 1791.567,A 0.000,B 0.000,C 90.000,E1 282.007} C_DIS
LIN {X -0.028,Y -388.575,Z 1791.563,A 0.000,B 0.000,C 90.000,E1 281.422} C_DIS
LIN {X 0.071,Y -387.394,Z 1791.560,A 0.000,B 0.000,C 90.000,E1 280.838} C_DIS
LIN {X 0.164,Y -385.837,Z 1791.557,A 0.000,B 0.000,C 90.000,E1 280.254} C_DIS
LIN {X -0.095,Y -382.889,Z 1791.552,A 0.000,B 0.000,C 90.000,E1 279.434} C_DIS
LIN {X -0.065,Y -379.234,Z 1791.547,A 0.000,B 0.000,C 90.000,E1 278.568} C_DIS
LIN {X -0.070,Y -374.760,Z 1791.543,A 0.000,B 0.000,C 90.000,E1 277.701} C_DIS
LIN {X -0.109,Y -369.417,Z 1791.538,A 0.000,B 0.000,C 90.000,E1 276.834} C_DIS
LIN {X 0.162,Y -363.113,Z 1791.533,A 0.000,B 0.000,C 90.000,E1 275.910} C_DIS
LIN {X 0.058,Y -358.190,Z 1791.530,A 0.000,B 0.000,C 90.000,E1 275.334} C_DIS
LIN {X -0.029,Y -352.720,Z 1791.526,A 0.000,B 0.000,C 90.000,E1 274.759} C_DIS
LIN {X 0.001,Y -346.957,Z 1791.523,A 0.000,B 0.000,C 90.000,E1 274.188} C_DIS
LIN {X -0.085,Y -341.050,Z 1791.520,A 0.000,B 0.000,C 90.000,E1 273.669} C_DIS
LIN {X 0.044,Y -334.991,Z 1791.518,A 0.000,B 0.000,C 90.000,E1 273.154} C_DIS
LIN {X 0.087,Y -328.748,Z 1791.515,A 0.000,B 0.000,C 90.000,E1 272.694} C_DIS
LIN {X -0.008,Y -322.312,Z 1791.513,A 0.000,B 0.000,C 90.000,E1 272.293} C_DIS
LIN {X 0.123,Y -315.611,Z 1791.511,A 0.000,B 0.000,C 90.000,E1 271.892} C_DIS
LIN {X -0.096,Y -308.548,Z 1791.509,A 0.000,B 0.000,C 90.000,E1 271.604} C_DIS
LIN {X -0.012,Y -301.004,Z 1791.507,A 0.000,B 0.000,C 90.000,E1 271.318} C_DIS
LIN {X -0.134,Y -289.623,Z 1791.506,A 0.000,B 0.000,C 90.000,E1 271.031} C_DIS
LIN {X 0.099,Y -278.895,Z 1791.504,A 0.000,B 0.000,C 90.000,E1 270.745} C_DIS
LIN {X -0.123,Y -263.042,Z 1791.503,A 0.000,B 0.000,C 90.000,E1 270.516} C_DIS
LIN {X 0.101,Y -254.225,Z 1791.502,A 0.000,B 0.000,C 90.000,E1 270.344} C_DIS
LIN {X 0.082,Y -238.455,Z 1791.501,A 0.000,B 0.000,C 90.000,E1 270.229} C_DIS
LIN {X 0.000,Y -230.900,Z 1791.501,A 0.000,B 0.000,C 90.000,E1 270.229} C_DIS
LIN {X -0.020,Y -181.580,Z 1791.501,A 0.000,B 0.000,C 90.000,E1 270.229} C_DIS
LIN {X -0.051,Y -180.811,Z 1791.471,A 0.000,B 0.000,C 90.000,E1 264.837} C_DIS
LIN {X 0.026,Y -178.914,Z 1791.443,A 0.000,B 0.000,C 90.000,E1 259.746} C_DIS
LIN {X -0.065,Y -175.958,Z 1791.415,A 0.000,B 0.000,C 90.000,E1 254.685} C_DIS
LIN {X 0.052,Y -175.431,Z 1791.410,A 0.000,B 0.000,C 90.000,E1 253.795} C_DIS
LIN {X 0.055,Y -172.190,Z 1791.386,A 0.000,B 0.000,C 90.000,E1 249.518} C_DIS
LIN {X 0.030,Y -171.663,Z 1791.382,A 0.000,B 0.000,C 90.000,E1 248.666} C_DIS
LIN {X 0.014,Y -167.887,Z 1791.358,A 0.000,B 0.000,C 90.000,E1 244.357} C_DIS
LIN {X 0.030,Y -166.624,Z 1791.348,A 0.000,B 0.000,C 90.000,E1 242.615} C_DIS
LIN {X 0.023,Y -162.611,Z 1791.324,A 0.000,B 0.000,C 90.000,E1 238.250} C_DIS
LIN {X -0.003,Y -161.297,Z 1791.314,A 0.000,B 0.000,C 90.000,E1 236.501} C_DIS
LIN {X 0.031,Y -157.294,Z 1791.289,A 0.000,B 0.000,C 90.000,E1 232.065} C_DIS
LIN {X 0.054,Y -156.011,Z 1791.279,A 0.000,B 0.000,C 90.000,E1 230.275} C_DIS
LIN {X 0.013,Y -152.270,Z 1791.255,A 0.000,B 0.000,C 90.000,E1 225.810} C_DIS
LIN {X 0.035,Y -150.506,Z 1791.240,A 0.000,B 0.000,C 90.000,E1 223.095} C_DIS
LIN {X 0.065,Y -147.230,Z 1791.214,A 0.000,B 0.000,C 90.000,E1 218.543} C_DIS
LIN {X 0.035,Y -145.254,Z 1791.194,A 0.000,B 0.000,C 90.000,E1 214.898} C_DIS
LIN {X -0.050,Y -142.368,Z 1791.163,A 0.000,B 0.000,C 90.000,E1 209.411} C_DIS
LIN {X 0.071,Y -141.753,Z 1791.153,A 0.000,B 0.000,C 90.000,E1 207.513} C_DIS
LIN {X -0.003,Y -139.495,Z 1791.117,A 0.000,B 0.000,C 90.000,E1 201.046} C_DIS
LIN {X 0.034,Y -139.001,Z 1791.101,A 0.000,B 0.000,C 90.000,E1 198.236} C_DIS
LIN {X -0.010,Y -138.338,Z 1791.055,A 0.000,B 0.000,C 90.000,E1 189.849} C_DIS
LIN {X 0.012,Y -139.410,Z 1791.008,A 0.000,B 0.000,C 90.000,E1 181.432} C_DIS
LIN {X 0.066,Y -141.320,Z 1790.972,A 0.000,B 0.000,C 90.000,E1 174.894} C_DIS
LIN {X 0.024,Y -142.679,Z 1790.956,A 0.000,B 0.000,C 90.000,E1 172.129} C_DIS
LIN {X 0.004,Y -145.035,Z 1790.931,A 0.000,B 0.000,C 90.000,E1 167.521} C_DIS
LIN {X -0.039,Y -147.661,Z 1790.910,A 0.000,B 0.000,C 90.000,E1 163.866} C_DIS
LIN {X 0.037,Y -150.300,Z 1790.890,A 0.000,B 0.000,C 90.000,E1 160.188} C_DIS
LIN {X -0.093,Y -153.709,Z 1790.870,A 0.000,B 0.000,C 90.000,E1 156.613} C_DIS
LIN {X -0.038,Y -157.123,Z 1790.850,A 0.000,B 0.000,C 90.000,E1 152.999} C_DIS
LIN {X 0.038,Y -161.267,Z 1790.830,A 0.000,B 0.000,C 90.000,E1 149.410} C_DIS
LIN {X -0.035,Y -164.385,Z 1790.815,A 0.000,B 0.000,C 90.000,E1 146.786} C_DIS
LIN {X -0.048,Y -169.062,Z 1790.796,A 0.000,B 0.000,C 90.000,E1 143.290} C_DIS
LIN {X 0.004,Y -171.622,Z 1790.786,A 0.000,B 0.000,C 90.000,E1 141.537} C_DIS
LIN {X 0.051,Y -176.579,Z 1790.767,A 0.000,B 0.000,C 90.000,E1 138.081} C_DIS
LIN {X -0.075,Y -180.878,Z 1790.753,A 0.000,B 0.000,C 90.000,E1 135.567} C_DIS
LIN {X 0.046,Y -186.291,Z 1790.734,A 0.000,B 0.000,C 90.000,E1 132.162} C_DIS
LIN {X 0.113,Y -190.926,Z 1790.720,A 0.000,B 0.000,C 90.000,E1 129.644} C_DIS
LIN {X 0.034,Y -196.694,Z 1790.702,A 0.000,B 0.000,C 90.000,E1 126.377} C_DIS
LIN {X 0.065,Y -199.938,Z 1790.693,A 0.000,B 0.000,C 90.000,E1 124.739} C_DIS
LIN {X -0.043,Y -205.855,Z 1790.675,A 0.000,B 0.000,C 90.000,E1 121.544} C_DIS
LIN {X -0.016,Y -210.871,Z 1790.661,A 0.000,B 0.000,C 90.000,E1 119.027} C_DIS
LIN {X -0.082,Y -211.391,Z 1790.660,A 0.000,B 0.000,C 90.000,E1 118.743} C_DIS
LIN {X 0.111,Y -338.202,Z 1790.660,A 0.000,B 0.000,C 90.000,E1 118.693} C_DIS
LIN {X -0.049,Y -339.893,Z 1790.659,A 0.000,B 0.000,C 90.000,E1 118.693} C_DIS
LIN {X 0.178,Y -343.863,Z 1790.658,A 0.000,B 0.000,C 90.000,E1 118.487} C_DIS
LIN {X -0.062,Y -346.120,Z 1790.657,A 0.000,B 0.000,C 90.000,E1 118.359} C_DIS
LIN {X 0.103,Y -349.885,Z 1790.655,A 0.000,B 0.000,C 90.000,E1 117.897} C_DIS
LIN {X 0.132,Y -351.654,Z 1790.653,A 0.000,B 0.000,C 90.000,E1 117.590} C_DIS
LIN {X -0.086,Y -360.691,Z 1790.642,A 0.000,B 0.000,C 90.000,E1 115.515} C_DIS
LIN {X 0.062,Y -372.604,Z 1790.627,A 0.000,B 0.000,C 90.000,E1 112.823} C_DIS
LIN {X -0.001,Y -381.961,Z 1790.615,A 0.000,B 0.000,C 90.000,E1 110.791} C_DIS
LIN {X 0.195,Y -388.425,Z 1790.608,A 0.000,B 0.000,C 90.000,E1 109.322} C_DIS
LIN {X 0.196,Y -393.179,Z 1790.601,A 0.000,B 0.000,C 90.000,E1 108.181} C_DIS
LIN {X 0.084,Y -396.182,Z 1790.596,A 0.000,B 0.000,C 90.000,E1 107.347} C_DIS
LIN {X -0.068,Y -397.602,Z 1790.593,A 0.000,B 0.000,C 90.000,E1 106.804} C_DIS
LIN {X 0.171,Y -397.819,Z 1790.590,A 0.000,B 0.000,C 90.000,E1 106.205} C_DIS
LIN {X 0.006,Y -392.056,Z 1790.556,A 0.000,B 0.000,C 90.000,E1 100.018} C_DIS
LIN {X 0.150,Y -391.392,Z 1790.547,A 0.000,B 0.000,C 90.000,E1 98.454} C_DIS
LIN {X 0.089,Y -391.428,Z 1790.547,A 0.000,B 0.000,C 90.000,E1 98.454} C_DIS
LIN {X -0.042,Y -412.325,Z 1790.537,A 0.000,B 0.000,C 90.000,E1 96.663} C_DIS
LIN {X -0.019,Y -434.755,Z 1790.527,A 0.000,B 0.000,C 90.000,E1 94.935} C_DIS
LIN {X 0.198,Y -437.603,Z 1790.526,A 0.000,B 0.000,C 90.000,E1 94.702} C_DIS
LIN {X 0.201,Y -441.987,Z 1790.524,A 0.000,B 0.000,C 90.000,E1 94.302} C_DIS
LIN {X 0.075,Y -445.083,Z 1790.521,A 0.000,B 0.000,C 90.000,E1 93.841} C_DIS
LIN {X -0.019,Y -447.049,Z 1790.518,A 0.000,B 0.000,C 90.000,E1 93.326} C_DIS
LIN {X -0.069,Y -447.921,Z 1790.516,A 0.000,B 0.000,C 90.000,E1 92.808} C_DIS
LIN {X -0.129,Y -447.854,Z 1790.513,A 0.000,B 0.000,C 90.000,E1 92.293} C_DIS
LIN {X -0.168,Y -446.841,Z 1790.510,A 0.000,B 0.000,C 90.000,E1 91.776} C_DIS
LIN {X 0.223,Y -444.718,Z 1790.507,A 0.000,B 0.000,C 90.000,E1 91.203} C_DIS
LIN {X -0.014,Y -434.873,Z 1790.498,A 0.000,B 0.000,C 90.000,E1 89.656} C_DIS
LIN {X 0.025,Y -424.945,Z 1790.489,A 0.000,B 0.000,C 90.000,E1 88.051} C_DIS
LIN {X -0.017,Y -413.170,Z 1790.479,A 0.000,B 0.000,C 90.000,E1 86.159} C_DIS
LIN {X 0.160,Y -401.281,Z 1790.468,A 0.000,B 0.000,C 90.000,E1 84.204} C_DIS
LIN {X 0.106,Y -399.851,Z 1790.467,A 0.000,B 0.000,C 90.000,E1 83.976} C_DIS
LIN {X 0.088,Y -399.851,Z 1790.467,A 0.000,B 0.000,C 90.000,E1 83.970} C_DIS
LIN {X -0.137,Y -403.125,Z 1790.455,A 0.000,B 0.000,C 90.000,E1 82.008} C_DIS
LIN {X -0.020,Y -402.765,Z 1790.452,A 0.000,B 0.000,C 90.000,E1 81.432} C_DIS
LIN {X 0.162,Y -401.588,Z 1790.449,A 0.000,B 0.000,C 90.000,E1 80.849} C_DIS
LIN {X -0.119,Y -400.037,Z 1790.446,A 0.000,B 0.000,C 90.000,E1 80.330} C_DIS
LIN {X -0.170,Y -396.346,Z 1790.440,A 0.000,B 0.000,C 90.000,E1 79.218} C_DIS
LIN {X 0.128,Y -392.210,Z 1790.434,A 0.000,B 0.000,C 90.000,E1 78.049} C_DIS
LIN {X 0.084,Y -385.556,Z 1790.424,A 0.000,B 0.000,C 90.000,E1 76.353} C_DIS
LIN {X 0.087,Y -378.602,Z 1790.415,A 0.000,B 0.000,C 90.000,E1 74.629} C_DIS
LIN {X 0.065,Y -370.343,Z 1790.403,A 0.000,B 0.000,C 90.000,E1 72.598} C_DIS
LIN {X -0.018,Y -361.916,Z 1790.392,A 0.000,B 0.000,C 90.000,E1 70.550} C_DIS
LIN {X 0.006,Y -352.130,Z 1790.379,A 0.000,B 0.000,C 90.000,E1 68.156} C_DIS
LIN {X -0.094,Y -343.466,Z 1790.367,A 0.000,B 0.000,C 90.000,E1 66.049} C_DIS
LIN {X -0.098,Y -334.697,Z 1790.355,A 0.000,B 0.000,C 90.000,E1 63.896} C_DIS
LIN {X 0.071,Y -328.202,Z 1790.346,A 0.000,B 0.000,C 90.000,E1 62.308} C_DIS
LIN {X 0.155,Y -321.318,Z 1790.338,A 0.000,B 0.000,C 90.000,E1 60.717} C_DIS
LIN {X 0.045,Y -312.638,Z 1790.327,A 0.000,B 0.000,C 90.000,E1 58.820} C_DIS
LIN {X -0.166,Y -303.690,Z 1790.316,A 0.000,B 0.000,C 90.000,E1 56.914} C_DIS
LIN {X 0.049,Y -293.160,Z 1790.303,A 0.000,B 0.000,C 90.000,E1 54.562} C_DIS
LIN {X 0.117,Y -278.639,Z 1790.284,A 0.000,B 0.000,C 90.000,E1 51.170} C_DIS
LIN {X -0.016,Y -266.492,Z 1790.267,A 0.000,B 0.000,C 90.000,E1 48.081} C_DIS
LIN {X 0.013,Y -256.322,Z 1790.251,A 0.000,B 0.000,C 90.000,E1 45.243} C_DIS
LIN {X -0.028,Y -245.439,Z 1790.233,A 0.000,B 0.000,C 90.000,E1 42.000} C_DIS
LIN {X 0.011,Y -235.043,Z 1790.215,A 0.000,B 0.000,C 90.000,E1 38.669} C_DIS
LIN {X -0.066,Y -226.265,Z 1790.198,A 0.000,B 0.000,C 90.000,E1 35.678} C_DIS
LIN {X -0.093,Y -217.964,Z 1790.181,A 0.000,B 0.000,C 90.000,E1 32.625} C_DIS
LIN {X -0.007,Y -210.302,Z 1790.164,A 0.000,B 0.000,C 90.000,E1 29.489} C_DIS
LIN {X 0.050,Y -203.269,Z 1790.146,A 0.000,B 0.000,C 90.000,E1 26.309} C_DIS
LIN {X 0.109,Y -197.030,Z 1790.128,A 0.000,B 0.000,C 90.000,E1 23.078} C_DIS
LIN {X -0.039,Y -191.657,Z 1790.110,A 0.000,B 0.000,C 90.000,E1 19.866} C_DIS
LIN {X 0.026,Y -187.190,Z 1790.092,A 0.000,B 0.000,C 90.000,E1 16.551} C_DIS
LIN {X -0.048,Y -182.877,Z 1790.069,A 0.000,B 0.000,C 90.000,E1 12.411} C_DIS
LIN {X -0.081,Y -179.628,Z 1790.046,A 0.000,B 0.000,C 90.000,E1 8.219} C_DIS
LIN {X 0.083,Y -176.824,Z 1790.013,A 0.000,B 0.000,C 90.000,E1 2.236} C_DIS
LIN {X -0.090,Y -175.805,Z 1789.974,A 0.000,B 0.000,C 90.000,E1 355.298} C_DIS
LIN {X 0.045,Y -176.443,Z 1789.941,A 0.000,B 0.000,C 90.000,E1 349.285} C_DIS
LIN {X 0.022,Y -178.756,Z 1789.903,A 0.000,B 0.000,C 90.000,E1 342.489} C_DIS
LIN {X 0.033,Y -181.776,Z 1789.875,A 0.000,B 0.000,C 90.000,E1 337.411} C_DIS
LIN {X 0.082,Y -185.638,Z 1789.847,A 0.000,B 0.000,C 90.000,E1 332.359} C_DIS
LIN {X 0.069,Y -189.649,Z 1789.823,A 0.000,B 0.000,C 90.000,E1 328.201} C_DIS
LIN {X -0.057,Y -194.696,Z 1789.801,A 0.000,B 0.000,C 90.000,E1 324.116} C_DIS
LIN {X 0.111,Y -199.719,Z 1789.782,A 0.000,B 0.000,C 90.000,E1 320.803} C_DIS
LIN {X -0.090,Y -206.003,Z 1789.765,A 0.000,B 0.000,C 90.000,E1 317.634} C_DIS
LIN {X -0.092,Y -211.587,Z 1789.751,A 0.000,B 0.000,C 90.000,E1 315.243} C_DIS
LIN {X -0.025,Y -216.991,Z 1789.740,A 0.000,B 0.000,C 90.000,E1 313.257} C_DIS
LIN {X 0.068,Y -221.963,Z 1789.732,A 0.000,B 0.000,C 90.000,E1 311.676} C_DIS
LIN {X -0.075,Y -227.623,Z 1789.723,A 0.000,B 0.000,C 90.000,E1 310.172} C_DIS
LIN {X -0.016,Y -235.710,Z 1789.713,A 0.000,B 0.000,C 90.000,E1 308.257} C_DIS
LIN {X 0.038,Y -244.919,Z 1789.702,A 0.000,B 0.000,C 90.000,E1 306.377} C_DIS
LIN {X -0.037,Y -257.128,Z 1789.690,A 0.000,B 0.000,C 90.000,E1 304.199} C_DIS
LIN {X 0.041,Y -275.166,Z 1789.674,A 0.000,B 0.000,C 90.000,E1 301.337} C_DIS
LIN {X -0.079,Y -294.743,Z 1789.659,A 0.000,B 0.000,C 90.000,E1 298.615} C_DIS
LIN {X -0.111,Y -315.433,Z 1789.644,A 0.000,B 0.000,C 90.000,E1 295.976} C_DIS
LIN {X 0.115,Y -328.605,Z 1789.635,A 0.000,B 0.000,C 90.000,E1 294.335} C_DIS
LIN {X 0.097,Y -341.430,Z 1789.627,A 0.000,B 0.000,C 90.000,E1 292.770} C_DIS
LIN {X 0.118,Y -351.463,Z 1789.620,A 0.000,B 0.000,C 90.000,E1 291.535} C_DIS
LIN {X -0.072,Y -361.009,Z 1789.613,A 0.000,B 0.000,C 90.000,E1 290.355} C_DIS
LIN {X -0.016,Y -367.650,Z 1789.608,A 0.000,B 0.000,C 90.000,E1 289.450} C_DIS
LIN {X 0.023,Y -371.703,Z 1789.605,A 0.000,B 0.000,C 90.000,E1 288.852} C_DIS
LIN {X 0.209,Y -375.377,Z 1789.601,A 0.000,B 0.000,C 90.000,E1 288.236} C_DIS
LIN {X -0.059,Y -378.577,Z 1789.598,A 0.000,B 0.000,C 90.000,E1 287.692} C_DIS
LIN {X 0.054,Y -381.370,Z 1789.595,A 0.000,B 0.000,C 90.000,E1 287.094} C_DIS
LIN {X 0.188,Y -383.755,Z 1789.592,A 0.000,B 0.000,C 90.000,E1 286.496} C_DIS
LIN {X -0.033,Y -385.747,Z 1789.589,A 0.000,B 0.000,C 90.000,E1 285.953} C_DIS
LIN {X 0.019,Y -387.419,Z 1789.585,A 0.000,B 0.000,C 90.000,E1 285.371} C_DIS
LIN {X 0.188,Y -388.721,Z 1789.582,A 0.000,B 0.000,C 90.000,E1 284.773} C_DIS
LIN {X -0.107,Y -389.669,Z 1789.579,A 0.000,B 0.000,C 90.000,E1 284.245} C_DIS
LIN {X 0.077,Y -390.215,Z 1789.576,A 0.000,B 0.000,C 90.000,E1 283.647} C_DIS
LIN {X 0.175,Y -390.428,Z 1789.573,A 0.000,B 0.000,C 90.000,E1 283.063} C_DIS
LIN {X -0.102,Y -390.280,Z 1789.570,A 0.000,B 0.000,C 90.000,E1 282.535} C_DIS
LIN {X 0.003,Y -389.777,Z 1789.566,A 0.000,B 0.000,C 90.000,E1 281.951} C_DIS
LIN {X 0.108,Y -388.921,Z 1789.563,A 0.000,B 0.000,C 90.000,E1 281.366} C_DIS
LIN {X -0.170,Y -387.693,Z 1789.560,A 0.000,B 0.000,C 90.000,E1 280.838} C_DIS
LIN {X -0.076,Y -386.125,Z 1789.557,A 0.000,B 0.000,C 90.000,E1 280.254} C_DIS
LIN {X 0.048,Y -383.133,Z 1789.552,A 0.000,B 0.000,C 90.000,E1 279.378} C_DIS
LIN {X 0.081,Y -379.419,Z 1789.547,A 0.000,B 0.000,C 90.000,E1 278.511} C_DIS
LIN {X 0.076,Y -374.900,Z 1789.542,A 0.000,B 0.000,C 90.000,E1 277.644} C_DIS
LIN {X 0.038,Y -369.499,Z 1789.538,A 0.000,B 0.000,C 90.000,E1 276.777} C_DIS
LIN {X -0.029,Y -365.391,Z 1789.534,A 0.000,B 0.000,C 90.000,E1 276.201} C_DIS
LIN {X -0.116,Y -360.726,Z 1789.531,A 0.000,B 0.000,C 90.000,E1 275.625} C_DIS
LIN {X 0.127,Y -355.446,Z 1789.528,A 0.000,B 0.000,C 90.000,E1 274.992} C_DIS
LIN {X 0.103,Y -349.771,Z 1789.525,A 0.000,B 0.000,C 90.000,E1 274.416} C_DIS
LIN {X -0.064,Y -343.892,Z 1789.522,A 0.000,B 0.000,C 90.000,E1 273.898} C_DIS
LIN {X -0.020,Y -337.906,Z 1789.519,A 0.000,B 0.000,C 90.000,E1 273.383} C_DIS
LIN {X -0.105,Y -331.663,Z 1789.516,A 0.000,B 0.000,C 90.000,E1 272.922} C_DIS
LIN {X 0.032,Y -325.264,Z 1789.514,A 0.000,B 0.000,C 90.000,E1 272.465} C_DIS
LIN {X 0.063,Y -318.649,Z 1789.511,A 0.000,B 0.000,C 90.000,E1 272.064} C_DIS
LIN {X 0.017,Y -311.638,Z 1789.510,A 0.000,B 0.000,C 90.000,E1 271.718} C_DIS
LIN {X -0.033,Y -304.240,Z 1789.508,A 0.000,B 0.000,C 90.000,E1 271.432} C_DIS
LIN {X -0.079,Y -296.556,Z 1789.507,A 0.000,B 0.000,C 90.000,E1 271.203} C_DIS
LIN {X 0.016,Y -285.891,Z 1789.505,A 0.000,B 0.000,C 90.000,E1 270.917} C_DIS
LIN {X 0.011,Y -274.751,Z 1789.504,A 0.000,B 0.000,C 90.000,E1 270.688} C_DIS
LIN {X 0.125,Y -258.471,Z 1789.502,A 0.000,B 0.000,C 90.000,E1 270.401} C_DIS
LIN {X 0.014,Y -244.463,Z 1789.502,A 0.000,B 0.000,C 90.000,E1 270.286} C_DIS
LIN {X 0.075,Y -234.777,Z 1789.501,A 0.000,B 0.000,C 90.000,E1 270.229} C_DIS
LIN {X 0.038,Y -181.581,Z 1789.501,A 0.000,B 0.000,C 90.000,E1 270.229} C_DIS
LIN {X -0.056,Y -180.891,Z 1789.473,A 0.000,B 0.000,C 90.000,E1 265.179} C_DIS
LIN {X 0.007,Y -179.016,Z 1789.445,A 0.000,B 0.000,C 90.000,E1 260.095} C_DIS
LIN {X 0.101,Y -178.642,Z 1789.440,A 0.000,B 0.000,C 90.000,E1 259.218} C_DIS
LIN {X -0.001,Y -175.693,Z 1789.412,A 0.000,B 0.000,C 90.000,E1 254.157} C_DIS
LIN {X 0.010,Y -172.409,Z 1789.388,A 0.000,B 0.000,C 90.000,E1 249.880} C_DIS
LIN {X 0.026,Y -171.224,Z 1789.379,A 0.000,B 0.000,C 90.000,E1 248.156} C_DIS
LIN {X 0.001,Y -167.505,Z 1789.355,A 0.000,B 0.000,C 90.000,E1 243.845} C_DIS
LIN {X -0.065,Y -166.901,Z 1789.350,A 0.000,B 0.000,C 90.000,E1 242.999} C_DIS
LIN {X -0.013,Y -162.209,Z 1789.321,A 0.000,B 0.000,C 90.000,E1 237.740} C_DIS
LIN {X 0.040,Y -160.785,Z 1789.311,A 0.000,B 0.000,C 90.000,E1 235.960} C_DIS
LIN {X 0.012,Y -157.577,Z 1789.291,A 0.000,B 0.000,C 90.000,E1 232.431} C_DIS
LIN {X 0.046,Y -155.608,Z 1789.276,A 0.000,B 0.000,C 90.000,E1 229.747} C_DIS
LIN {X -0.011,Y -151.888,Z 1789.252,A 0.000,B 0.000,C 90.000,E1 225.283} C_DIS
LIN {X 0.008,Y -150.115,Z 1789.236,A 0.000,B 0.000,C 90.000,E1 222.567} C_DIS
LIN {X 0.026,Y -146.909,Z 1789.211,A 0.000,B 0.000,C 90.000,E1 218.016} C_DIS
LIN {X -0.073,Y -145.497,Z 1789.196,A 0.000,B 0.000,C 90.000,E1 215.311} C_DIS
LIN {X 0.045,Y -142.902,Z 1789.171,A 0.000,B 0.000,C 90.000,E1 210.669} C_DIS
LIN {X -0.025,Y -141.522,Z 1789.150,A 0.000,B 0.000,C 90.000,E1 207.001} C_DIS
LIN {X 0.019,Y -139.395,Z 1789.114,A 0.000,B 0.000,C 90.000,E1 200.482} C_DIS
LIN {X 0.070,Y -139.107,Z 1789.104,A 0.000,B 0.000,C 90.000,E1 198.598} C_DIS
LIN {X 0.061,Y -138.353,Z 1789.057,A 0.000,B 0.000,C 90.000,E1 190.197} C_DIS
LIN {X 0.055,Y -139.511,Z 1789.005,A 0.000,B 0.000,C 90.000,E1 180.859} C_DIS
LIN {X -0.005,Y -141.153,Z 1788.974,A 0.000,B 0.000,C 90.000,E1 175.298} C_DIS
LIN {X -0.034,Y -142.533,Z 1788.958,A 0.000,B 0.000,C 90.000,E1 172.527} C_DIS
LIN {X 0.034,Y -144.803,Z 1788.933,A 0.000,B 0.000,C 90.000,E1 167.881} C_DIS
LIN {X 0.023,Y -147.421,Z 1788.912,A 0.000,B 0.000,C 90.000,E1 164.212} C_DIS
LIN {X 0.052,Y -149.998,Z 1788.892,A 0.000,B 0.000,C 90.000,E1 160.550} C_DIS
LIN {X 0.059,Y -153.328,Z 1788.872,A 0.000,B 0.000,C 90.000,E1 156.922} C_DIS
LIN {X -0.029,Y -155.027,Z 1788.862,A 0.000,B 0.000,C 90.000,E1 155.153} C_DIS
LIN {X -0.008,Y -158.675,Z 1788.842,A 0.000,B 0.000,C 90.000,E1 151.563} C_DIS
LIN {X 0.075,Y -161.953,Z 1788.827,A 0.000,B 0.000,C 90.000,E1 148.869} C_DIS
LIN {X -0.041,Y -166.145,Z 1788.808,A 0.000,B 0.000,C 90.000,E1 145.388} C_DIS
LIN {X -0.045,Y -171.157,Z 1788.788,A 0.000,B 0.000,C 90.000,E1 141.904} C_DIS
LIN {X -0.011,Y -176.036,Z 1788.769,A 0.000,B 0.000,C 90.000,E1 138.447} C_DIS
LIN {X -0.014,Y -180.290,Z 1788.755,A 0.000,B 0.000,C 90.000,E1 135.891} C_DIS
LIN {X -0.042,Y -185.702,Z 1788.736,A 0.000,B 0.000,C 90.000,E1 132.528} C_DIS
LIN {X 0.009,Y -190.308,Z 1788.722,A 0.000,B 0.000,C 90.000,E1 130.011} C_DIS
LIN {X 0.057,Y -197.634,Z 1788.699,A 0.000,B 0.000,C 90.000,E1 125.884} C_DIS
LIN {X -0.014,Y -200.891,Z 1788.690,A 0.000,B 0.000,C 90.000,E1 124.278} C_DIS
LIN {X 0.012,Y -206.793,Z 1788.672,A 0.000,B 0.000,C 90.000,E1 121.052} C_DIS
LIN {X -0.021,Y -210.705,Z 1788.662,A 0.000,B 0.000,C 90.000,E1 119.127} C_DIS
LIN {X -0.027,Y -211.231,Z 1788.660,A 0.000,B 0.000,C 90.000,E1 118.821} C_DIS
LIN {X -0.078,Y -338.023,Z 1788.660,A 0.000,B 0.000,C 90.000,E1 118.821} C_DIS
LIN {X -0.184,Y -339.405,Z 1788.660,A 0.000,B 0.000,C 90.000,E1 118.821} C_DIS
LIN {X -0.144,Y -342.912,Z 1788.659,A 0.000,B 0.000,C 90.000,E1 118.693} C_DIS
LIN {X 0.095,Y -346.138,Z 1788.658,A 0.000,B 0.000,C 90.000,E1 118.437} C_DIS
LIN {X 0.178,Y -349.772,Z 1788.656,A 0.000,B 0.000,C 90.000,E1 118.025} C_DIS
LIN {X -0.039,Y -351.613,Z 1788.654,A 0.000,B 0.000,C 90.000,E1 117.769} C_DIS
LIN {X -0.041,Y -355.653,Z 1788.649,A 0.000,B 0.000,C 90.000,E1 116.873} C_DIS
LIN {X -0.126,Y -369.236,Z 1788.633,A 0.000,B 0.000,C 90.000,E1 113.898} C_DIS
LIN {X 0.008,Y -380.552,Z 1788.620,A 0.000,B 0.000,C 90.000,E1 111.535} C_DIS
LIN {X 0.124,Y -390.530,Z 1788.608,A 0.000,B 0.000,C 90.000,E1 109.504} C_DIS
LIN {X -0.056,Y -397.443,Z 1788.601,A 0.000,B 0.000,C 90.000,E1 108.109} C_DIS
LIN {X -0.065,Y -402.555,Z 1788.594,A 0.000,B 0.000,C 90.000,E1 106.985} C_DIS
LIN {X -0.178,Y -404.822,Z 1788.591,A 0.000,B 0.000,C 90.000,E1 106.441} C_DIS
LIN {X 0.111,Y -406.725,Z 1788.588,A 0.000,B 0.000,C 90.000,E1 105.843} C_DIS
LIN {X 0.014,Y -407.933,Z 1788.585,A 0.000,B 0.000,C 90.000,E1 105.300} C_DIS
LIN {X -0.180,Y -407.642,Z 1788.582,A 0.000,B 0.000,C 90.000,E1 104.773} C_DIS
LIN {X 0.055,Y -402.638,Z 1788.542,A 0.000,B 0.000,C 90.000,E1 97.466} C_DIS
LIN {X -0.006,Y -402.687,Z 1788.542,A 0.000,B 0.000,C 90.000,E1 97.466} C_DIS
LIN {X 0.011,Y -425.404,Z 1788.531,A 0.000,B 0.000,C 90.000,E1 95.625} C_DIS
LIN {X 0.040,Y -439.370,Z 1788.526,A 0.000,B 0.000,C 90.000,E1 94.588} C_DIS
LIN {X -0.184,Y -441.426,Z 1788.524,A 0.000,B 0.000,C 90.000,E1 94.416} C_DIS
LIN {X 0.094,Y -443.372,Z 1788.523,A 0.000,B 0.000,C 90.000,E1 94.131} C_DIS
LIN {X -0.038,Y -444.856,Z 1788.522,A 0.000,B 0.000,C 90.000,E1 93.898} C_DIS
LIN {X 0.141,Y -446.044,Z 1788.520,A 0.000,B 0.000,C 90.000,E1 93.612} C_DIS
LIN {X -0.124,Y -446.919,Z 1788.519,A 0.000,B 0.000,C 90.000,E1 93.383} C_DIS
LIN {X -0.169,Y -447.871,Z 1788.516,A 0.000,B 0.000,C 90.000,E1 92.865} C_DIS
LIN {X 0.216,Y -447.880,Z 1788.513,A 0.000,B 0.000,C 90.000,E1 92.293} C_DIS
LIN {X 0.177,Y -446.949,Z 1788.510,A 0.000,B 0.000,C 90.000,E1 91.776} C_DIS
LIN {X 0.122,Y -444.931,Z 1788.507,A 0.000,B 0.000,C 90.000,E1 91.260} C_DIS
LIN {X -0.014,Y -438.433,Z 1788.501,A 0.000,B 0.000,C 90.000,E1 90.229} C_DIS
LIN {X -0.214,Y -426.881,Z 1788.491,A 0.000,B 0.000,C 90.000,E1 88.396} C_DIS
LIN {X -0.189,Y -415.114,Z 1788.480,A 0.000,B 0.000,C 90.000,E1 86.502} C_DIS
LIN {X 0.121,Y -409.365,Z 1788.475,A 0.000,B 0.000,C 90.000,E1 85.527} C_DIS
LIN {X 0.059,Y -409.327,Z 1788.475,A 0.000,B 0.000,C 90.000,E1 85.527} C_DIS
LIN {X -0.134,Y -412.012,Z 1788.465,A 0.000,B 0.000,C 90.000,E1 83.742} C_DIS
LIN {X 0.044,Y -412.356,Z 1788.462,A 0.000,B 0.000,C 90.000,E1 83.166} C_DIS
LIN {X -0.185,Y -411.423,Z 1788.459,A 0.000,B 0.000,C 90.000,E1 82.648} C_DIS
LIN {X 0.052,Y -409.958,Z 1788.456,A 0.000,B 0.000,C 90.000,E1 82.064} C_DIS
LIN {X -0.177,Y -408.190,Z 1788.453,A 0.000,B 0.000,C 90.000,E1 81.546} C_DIS
LIN {X 0.199,Y -404.142,Z 1788.447,A 0.000,B 0.000,C 90.000,E1 80.387} C_DIS
LIN {X -0.101,Y -397.437,Z 1788.438,A 0.000,B 0.000,C 90.000,E1 78.757} C_DIS
LIN {X -0.065,Y -390.322,Z 1788.428,A 0.000,B 0.000,C 90.000,E1 77.061} C_DIS
LIN {X 0.053,Y -381.795,Z 1788.417,A 0.000,B 0.000,C 90.000,E1 75.046} C_DIS
LIN {X 0.100,Y -373.161,Z 1788.406,A 0.000,B 0.000,C 90.000,E1 73.015} C_DIS
LIN {X 0.073,Y -364.449,Z 1788.394,A 0.000,B 0.000,C 90.000,E1 70.967} C_DIS
LIN {X -0.020,Y -355.575,Z 1788.383,A 0.000,B 0.000,C 90.000,E1 68.901} C_DIS
LIN {X -0.049,Y -346.673,Z 1788.371,A 0.000,B 0.000,C 90.000,E1 66.794} C_DIS
LIN {X -0.128,Y -337.643,Z 1788.359,A 0.000,B 0.000,C 90.000,E1 64.665} C_DIS
LIN {X -0.080,Y -329.755,Z 1788.349,A 0.000,B 0.000,C 90.000,E1 62.794} C_DIS
LIN {X -0.177,Y -321.587,Z 1788.338,A 0.000,B 0.000,C 90.000,E1 60.923} C_DIS
LIN {X 0.084,Y -314.415,Z 1788.329,A 0.000,B 0.000,C 90.000,E1 59.282} C_DIS
LIN {X -0.095,Y -305.544,Z 1788.319,A 0.000,B 0.000,C 90.000,E1 57.375} C_DIS
LIN {X -0.009,Y -296.511,Z 1788.308,A 0.000,B 0.000,C 90.000,E1 55.388} C_DIS
LIN {X -0.002,Y -281.791,Z 1788.289,A 0.000,B 0.000,C 90.000,E1 52.029} C_DIS
LIN {X -0.011,Y -269.384,Z 1788.272,A 0.000,B 0.000,C 90.000,E1 48.933} C_DIS
LIN {X 0.130,Y -257.830,Z 1788.254,A 0.000,B 0.000,C 90.000,E1 45.729} C_DIS
LIN {X -0.053,Y -246.797,Z 1788.236,A 0.000,B 0.000,C 90.000,E1 42.528} C_DIS
LIN {X 0.019,Y -236.300,Z 1788.218,A 0.000,B 0.000,C 90.000,E1 39.197} C_DIS
LIN {X 0.061,Y -226.364,Z 1788.199,A 0.000,B 0.000,C 90.000,E1 35.804} C_DIS
LIN {X 0.030,Y -218.013,Z 1788.182,A 0.000,B 0.000,C 90.000,E1 32.752} C_DIS
LIN {X -0.073,Y -210.329,Z 1788.165,A 0.000,B 0.000,C 90.000,E1 29.667} C_DIS
LIN {X -0.020,Y -203.251,Z 1788.147,A 0.000,B 0.000,C 90.000,E1 26.488} C_DIS
LIN {X 0.038,Y -196.963,Z 1788.129,A 0.000,B 0.000,C 90.000,E1 23.259} C_DIS
LIN {X 0.068,Y -191.540,Z 1788.111,A 0.000,B 0.000,C 90.000,E1 19.993} C_DIS
LIN {X -0.049,Y -187.019,Z 1788.093,A 0.000,B 0.000,C 90.000,E1 16.732} C_DIS
LIN {X 0.056,Y -182.654,Z 1788.070,A 0.000,B 0.000,C 90.000,E1 12.535} C_DIS
LIN {X 0.022,Y -179.391,Z 1788.046,A 0.000,B 0.000,C 90.000,E1 8.341} C_DIS
LIN {X -0.015,Y -176.818,Z 1788.018,A 0.000,B 0.000,C 90.000,E1 3.269} C_DIS
LIN {X 0.053,Y -175.509,Z 1787.978,A 0.000,B 0.000,C 90.000,E1 356.102} C_DIS
LIN {X -0.019,Y -175.961,Z 1787.945,A 0.000,B 0.000,C 90.000,E1 350.151} C_DIS
LIN {X 0.030,Y -178.053,Z 1787.907,A 0.000,B 0.000,C 90.000,E1 343.323} C_DIS
LIN {X 0.059,Y -180.932,Z 1787.879,A 0.000,B 0.000,C 90.000,E1 338.230} C_DIS
LIN {X -0.008,Y -184.659,Z 1787.851,A 0.000,B 0.000,C 90.000,E1 333.204} C_DIS
LIN {X 0.110,Y -188.572,Z 1787.828,A 0.000,B 0.000,C 90.000,E1 328.997} C_DIS
LIN {X 0.006,Y -193.428,Z 1787.805,A 0.000,B 0.000,C 90.000,E1 324.895} C_DIS
LIN {X 0.023,Y -198.305,Z 1787.787,A 0.000,B 0.000,C 90.000,E1 321.618} C_DIS
LIN {X 0.062,Y -202.724,Z 1787.773,A 0.000,B 0.000,C 90.000,E1 319.175} C_DIS
LIN {X 0.008,Y -207.824,Z 1787.760,A 0.000,B 0.000,C 90.000,E1 316.782} C_DIS
LIN {X -0.103,Y -213.782,Z 1787.747,A 0.000,B 0.000,C 90.000,E1 314.433} C_DIS
LIN {X 0.006,Y -219.562,Z 1787.736,A 0.000,B 0.000,C 90.000,E1 312.447} C_DIS
LIN {X -0.020,Y -224.906,Z 1787.727,A 0.000,B 0.000,C 90.000,E1 310.906} C_DIS
LIN {X 0.048,Y -230.956,Z 1787.719,A 0.000,B 0.000,C 90.000,E1 309.358} C_DIS
LIN {X 0.012,Y -237.721,Z 1787.710,A 0.000,B 0.000,C 90.000,E1 307.855} C_DIS
LIN {X -0.059,Y -247.165,Z 1787.700,A 0.000,B 0.000,C 90.000,E1 306.011} C_DIS
LIN {X 0.117,Y -259.613,Z 1787.688,A 0.000,B 0.000,C 90.000,E1 303.785} C_DIS
LIN {X -0.109,Y -277.878,Z 1787.672,A 0.000,B 0.000,C 90.000,E1 301.003} C_DIS
LIN {X 0.106,Y -295.143,Z 1787.659,A 0.000,B 0.000,C 90.000,E1 298.565} C_DIS
LIN {X 0.107,Y -315.866,Z 1787.644,A 0.000,B 0.000,C 90.000,E1 295.924} C_DIS
LIN {X 0.045,Y -329.081,Z 1787.635,A 0.000,B 0.000,C 90.000,E1 294.335} C_DIS
LIN {X 0.041,Y -339.388,Z 1787.628,A 0.000,B 0.000,C 90.000,E1 293.078} C_DIS
LIN {X 0.057,Y -351.944,Z 1787.620,A 0.000,B 0.000,C 90.000,E1 291.535} C_DIS
LIN {X -0.129,Y -361.537,Z 1787.613,A 0.000,B 0.000,C 90.000,E1 290.355} C_DIS
LIN {X -0.069,Y -368.184,Z 1787.608,A 0.000,B 0.000,C 90.000,E1 289.450} C_DIS
LIN {X -0.027,Y -372.231,Z 1787.605,A 0.000,B 0.000,C 90.000,E1 288.852} C_DIS
LIN {X 0.162,Y -375.882,Z 1787.601,A 0.000,B 0.000,C 90.000,E1 288.236} C_DIS
LIN {X -0.103,Y -379.073,Z 1787.598,A 0.000,B 0.000,C 90.000,E1 287.692} C_DIS
LIN {X 0.012,Y -381.892,Z 1787.595,A 0.000,B 0.000,C 90.000,E1 287.094} C_DIS
LIN {X 0.149,Y -384.210,Z 1787.592,A 0.000,B 0.000,C 90.000,E1 286.496} C_DIS
LIN {X -0.069,Y -386.197,Z 1787.589,A 0.000,B 0.000,C 90.000,E1 285.953} C_DIS
LIN {X -0.014,Y -387.868,Z 1787.585,A 0.000,B 0.000,C 90.000,E1 285.371} C_DIS
LIN {X 0.157,Y -389.155,Z 1787.582,A 0.000,B 0.000,C 90.000,E1 284.773} C_DIS
LIN {X -0.136,Y -390.093,Z 1787.579,A 0.000,B 0.000,C 90.000,E1 284.245} C_DIS
LIN {X 0.052,Y -390.638,Z 1787.576,A 0.000,B 0.000,C 90.000,E1 283.647} C_DIS
LIN {X 0.152,Y -390.822,Z 1787.573,A 0.000,B 0.000,C 90.000,E1 283.063} C_DIS
LIN {X -0.123,Y -390.654,Z 1787.570,A 0.000,B 0.000,C 90.000,E1 282.535} C_DIS
LIN {X -0.016,Y -390.157,Z 1787.566,A 0.000,B 0.000,C 90.000,E1 281.951} C_DIS
LIN {X 0.093,Y -389.298,Z 1787.563,A 0.000,B 0.000,C 90.000,E1 281.366} C_DIS
LIN {X -0.185,Y -388.081,Z 1787.560,A 0.000,B 0.000,C 90.000,E1 280.838} C_DIS
LIN {X -0.086,Y -386.510,Z 1787.557,A 0.000,B 0.000,C 90.000,E1 280.254} C_DIS
LIN {X 0.041,Y -383.508,Z 1787.552,A 0.000,B 0.000,C 90.000,E1 279.378} C_DIS
LIN {X 0.076,Y -379.775,Z 1787.547,A 0.000,B 0.000,C 90.000,E1 278.511} C_DIS
LIN {X 0.075,Y -375.237,Z 1787.542,A 0.000,B 0.000,C 90.000,E1 277.644} C_DIS
LIN {X 0.039,Y -369.804,Z 1787.538,A 0.000,B 0.000,C 90.000,E1 276.777} C_DIS
LIN {X -0.025,Y -365.687,Z 1787.534,A 0.000,B 0.000,C 90.000,E1 276.201} C_DIS
LIN {X -0.111,Y -360.988,Z 1787.531,A 0.000,B 0.000,C 90.000,E1 275.625} C_DIS
LIN {X 0.133,Y -355.734,Z 1787.528,A 0.000,B 0.000,C 90.000,E1 274.992} C_DIS
LIN {X 0.106,Y -350.013,Z 1787.525,A 0.000,B 0.000,C 90.000,E1 274.416} C_DIS
LIN {X -0.050,Y -344.115,Z 1787.522,A 0.000,B 0.000,C 90.000,E1 273.898} C_DIS
LIN {X -0.032,Y -335.111,Z 1787.517,A 0.000,B 0.000,C 90.000,E1 273.154} C_DIS
LIN {X 0.005,Y -328.800,Z 1787.515,A 0.000,B 0.000,C 90.000,E1 272.694} C_DIS
LIN {X -0.074,Y -322.221,Z 1787.513,A 0.000,B 0.000,C 90.000,E1 272.293} C_DIS
LIN {X 0.087,Y -315.516,Z 1787.511,A 0.000,B 0.000,C 90.000,E1 271.892} C_DIS
LIN {X -0.104,Y -308.305,Z 1787.509,A 0.000,B 0.000,C 90.000,E1 271.604} C_DIS
LIN {X -0.002,Y -300.817,Z 1787.507,A 0.000,B 0.000,C 90.000,E1 271.318} C_DIS
LIN {X -0.086,Y -289.670,Z 1787.506,A 0.000,B 0.000,C 90.000,E1 271.031} C_DIS
LIN {X -0.123,Y -278.856,Z 1787.504,A 0.000,B 0.000,C 90.000,E1 270.802} C_DIS
LIN {X -0.039,Y -263.411,Z 1787.503,A 0.000,B 0.000,C 90.000,E1 270.516} C_DIS
LIN {X -0.069,Y -254.189,Z 1787.502,A 0.000,B 0.000,C 90.000,E1 270.401} C_DIS
LIN {X 0.076,Y -245.140,Z 1787.502,A 0.000,B 0.000,C 90.000,E1 270.286} C_DIS
LIN {X -0.103,Y -235.581,Z 1787.501,A 0.000,B 0.000,C 90.000,E1 270.286} C_DIS
LIN {X 0.103,Y -229.746,Z 1787.501,A 0.000,B 0.000,C 90.000,E1 270.229} C_DIS
LIN {X 0.060,Y -181.581,Z 1787.501,A 0.000,B 0.000,C 90.000,E1 270.229} C_DIS
LIN {X 0.007,Y -180.818,Z 1787.471,A 0.000,B 0.000,C 90.000,E1 264.837} C_DIS
LIN {X 0.083,Y -178.921,Z 1787.443,A 0.000,B 0.000,C 90.000,E1 259.746} C_DIS
LIN {X -0.008,Y -175.966,Z 1787.415,A 0.000,B 0.000,C 90.000,E1 254.685} C_DIS
LIN {X -0.060,Y -175.446,Z 1787.410,A 0.000,B 0.000,C 90.000,E1 253.850} C_DIS
LIN {X -0.051,Y -172.201,Z 1787.386,A 0.000,B 0.000,C 90.000,E1 249.571} C_DIS
LIN {X -0.073,Y -171.676,Z 1787.382,A 0.000,B 0.000,C 90.000,E1 248.720} C_DIS
